   // === Motion positions (generated from XML) START ===
   ACTUAL_CHOOSEN_TYPE.Motion.Gluing_Nozzle_Z.Position[1].Pos := 143.76;
   ACTUAL_CHOOSEN_TYPE.Motion.Gluing_Nozzle_Z.Position[1].Vel := 200;
   ACTUAL_CHOOSEN_TYPE.Motion.Gluing_Nozzle_Z.Position[2].Pos := 139.11;
   ACTUAL_CHOOSEN_TYPE.Motion.Gluing_Nozzle_Z.Position[2].Vel := 200;
   ACTUAL_CHOOSEN_TYPE.Motion.Gluing_Nozzle_Z.Position[3].Pos := 131.98;
   ACTUAL_CHOOSEN_TYPE.Motion.Gluing_Nozzle_Z.Position[3].Vel := 200;
   ACTUAL_CHOOSEN_TYPE.Motion.Gluing_Nozzle_Z.Position[4].Pos := 127.89;
   ACTUAL_CHOOSEN_TYPE.Motion.Gluing_Nozzle_Z.Position[4].Vel := 200;
   ACTUAL_CHOOSEN_TYPE.Motion.Gluing_Nozzle_Z.Position[5].Pos := 0.0;
   ACTUAL_CHOOSEN_TYPE.Motion.Gluing_Nozzle_Z.Position[5].Vel := 0;
   ACTUAL_CHOOSEN_TYPE.Motion.Gluing_Nozzle_Z.Position[6].Pos := 127.0;
   ACTUAL_CHOOSEN_TYPE.Motion.Gluing_Nozzle_Z.Position[6].Vel := 200;
   ACTUAL_CHOOSEN_TYPE.Motion.Gluing_Nozzle_Z.Position[7].Pos := 48.11;
   ACTUAL_CHOOSEN_TYPE.Motion.Gluing_Nozzle_Z.Position[7].Vel := 200;
   ACTUAL_CHOOSEN_TYPE.Motion.Gluing_Nozzle_Z.Position[8].Pos := 0.0;
   ACTUAL_CHOOSEN_TYPE.Motion.Gluing_Nozzle_Z.Position[8].Vel := 200;
   ACTUAL_CHOOSEN_TYPE.Motion.Gluing_Nozzle_Z.Position[9].Pos := 123.0;
   ACTUAL_CHOOSEN_TYPE.Motion.Gluing_Nozzle_Z.Position[9].Vel := 200;
   ACTUAL_CHOOSEN_TYPE.Motion.Gluing_Nozzle_Z.Position[10].Pos := 0.0;
   ACTUAL_CHOOSEN_TYPE.Motion.Gluing_Nozzle_Z.Position[10].Vel := 0;
   ACTUAL_CHOOSEN_TYPE.Motion.Gluing_Nozzle_Z.Position[11].Pos := 0.0;
   ACTUAL_CHOOSEN_TYPE.Motion.Gluing_Nozzle_Z.Position[11].Vel := 0;
   ACTUAL_CHOOSEN_TYPE.Motion.Gluing_Nozzle_Z.Position[12].Pos := 0.0;
   ACTUAL_CHOOSEN_TYPE.Motion.Gluing_Nozzle_Z.Position[12].Vel := 0;
   ACTUAL_CHOOSEN_TYPE.Motion.Gluing_Nozzle_Z.Position[13].Pos := 0.0;
   ACTUAL_CHOOSEN_TYPE.Motion.Gluing_Nozzle_Z.Position[13].Vel := 0;
   ACTUAL_CHOOSEN_TYPE.Motion.Gluing_Nozzle_Z.Position[14].Pos := 0.0;
   ACTUAL_CHOOSEN_TYPE.Motion.Gluing_Nozzle_Z.Position[14].Vel := 0;
   ACTUAL_CHOOSEN_TYPE.Motion.Gluing_Nozzle_Z.Position[15].Pos := 0.0;
   ACTUAL_CHOOSEN_TYPE.Motion.Gluing_Nozzle_Z.Position[15].Vel := 0;
   ACTUAL_CHOOSEN_TYPE.Motion.Gluing_Nozzle_Z.Position[16].Pos := 0.0;
   ACTUAL_CHOOSEN_TYPE.Motion.Gluing_Nozzle_Z.Position[16].Vel := 0;
   ACTUAL_CHOOSEN_TYPE.Motion.Gluing_Nozzle_Z.Position[17].Pos := 0.0;
   ACTUAL_CHOOSEN_TYPE.Motion.Gluing_Nozzle_Z.Position[17].Vel := 0;
   ACTUAL_CHOOSEN_TYPE.Motion.Gluing_Nozzle_Z.Position[18].Pos := 0.0;
   ACTUAL_CHOOSEN_TYPE.Motion.Gluing_Nozzle_Z.Position[18].Vel := 0;
   ACTUAL_CHOOSEN_TYPE.Motion.Gluing_Nozzle_Z.Position[19].Pos := 0.0;
   ACTUAL_CHOOSEN_TYPE.Motion.Gluing_Nozzle_Z.Position[19].Vel := 0;
   ACTUAL_CHOOSEN_TYPE.Motion.Gluing_Nozzle_Z.Position[20].Pos := 0.0;
   ACTUAL_CHOOSEN_TYPE.Motion.Gluing_Nozzle_Z.Position[20].Vel := 0;
   ACTUAL_CHOOSEN_TYPE.Motion.Gluing_Nozzle_X.Position[1].Pos := 2.34;
   ACTUAL_CHOOSEN_TYPE.Motion.Gluing_Nozzle_X.Position[1].Vel := 200;
   ACTUAL_CHOOSEN_TYPE.Motion.Gluing_Nozzle_X.Position[2].Pos := 76.0;
   ACTUAL_CHOOSEN_TYPE.Motion.Gluing_Nozzle_X.Position[2].Vel := 200;
   ACTUAL_CHOOSEN_TYPE.Motion.Gluing_Nozzle_X.Position[3].Pos := 84.69;
   ACTUAL_CHOOSEN_TYPE.Motion.Gluing_Nozzle_X.Position[3].Vel := 200;
   ACTUAL_CHOOSEN_TYPE.Motion.Gluing_Nozzle_X.Position[4].Pos := 84.69;
   ACTUAL_CHOOSEN_TYPE.Motion.Gluing_Nozzle_X.Position[4].Vel := 200;
   ACTUAL_CHOOSEN_TYPE.Motion.Gluing_Nozzle_X.Position[5].Pos := 84.69;
   ACTUAL_CHOOSEN_TYPE.Motion.Gluing_Nozzle_X.Position[5].Vel := 200;
   ACTUAL_CHOOSEN_TYPE.Motion.Gluing_Nozzle_X.Position[6].Pos := 84.69;
   ACTUAL_CHOOSEN_TYPE.Motion.Gluing_Nozzle_X.Position[6].Vel := 200;
   ACTUAL_CHOOSEN_TYPE.Motion.Gluing_Nozzle_X.Position[7].Pos := 85.0;
   ACTUAL_CHOOSEN_TYPE.Motion.Gluing_Nozzle_X.Position[7].Vel := 200;
   ACTUAL_CHOOSEN_TYPE.Motion.Gluing_Nozzle_X.Position[8].Pos := 88.53;
   ACTUAL_CHOOSEN_TYPE.Motion.Gluing_Nozzle_X.Position[8].Vel := 200;
   ACTUAL_CHOOSEN_TYPE.Motion.Gluing_Nozzle_X.Position[9].Pos := 0.0;
   ACTUAL_CHOOSEN_TYPE.Motion.Gluing_Nozzle_X.Position[9].Vel := 0;
   ACTUAL_CHOOSEN_TYPE.Motion.Gluing_Nozzle_X.Position[10].Pos := 0.0;
   ACTUAL_CHOOSEN_TYPE.Motion.Gluing_Nozzle_X.Position[10].Vel := 0;
   ACTUAL_CHOOSEN_TYPE.Motion.Gluing_Nozzle_X.Position[11].Pos := 0.0;
   ACTUAL_CHOOSEN_TYPE.Motion.Gluing_Nozzle_X.Position[11].Vel := 0;
   ACTUAL_CHOOSEN_TYPE.Motion.Gluing_Nozzle_X.Position[12].Pos := 0.0;
   ACTUAL_CHOOSEN_TYPE.Motion.Gluing_Nozzle_X.Position[12].Vel := 0;
   ACTUAL_CHOOSEN_TYPE.Motion.Gluing_Nozzle_X.Position[13].Pos := 0.0;
   ACTUAL_CHOOSEN_TYPE.Motion.Gluing_Nozzle_X.Position[13].Vel := 0;
   ACTUAL_CHOOSEN_TYPE.Motion.Gluing_Nozzle_X.Position[14].Pos := 0.0;
   ACTUAL_CHOOSEN_TYPE.Motion.Gluing_Nozzle_X.Position[14].Vel := 0;
   ACTUAL_CHOOSEN_TYPE.Motion.Gluing_Nozzle_X.Position[15].Pos := 0.0;
   ACTUAL_CHOOSEN_TYPE.Motion.Gluing_Nozzle_X.Position[15].Vel := 0;
   ACTUAL_CHOOSEN_TYPE.Motion.Gluing_Nozzle_X.Position[16].Pos := 0.0;
   ACTUAL_CHOOSEN_TYPE.Motion.Gluing_Nozzle_X.Position[16].Vel := 0;
   ACTUAL_CHOOSEN_TYPE.Motion.Gluing_Nozzle_X.Position[17].Pos := 0.0;
   ACTUAL_CHOOSEN_TYPE.Motion.Gluing_Nozzle_X.Position[17].Vel := 0;
   ACTUAL_CHOOSEN_TYPE.Motion.Gluing_Nozzle_X.Position[18].Pos := 0.0;
   ACTUAL_CHOOSEN_TYPE.Motion.Gluing_Nozzle_X.Position[18].Vel := 0;
   ACTUAL_CHOOSEN_TYPE.Motion.Gluing_Nozzle_X.Position[19].Pos := 0.0;
   ACTUAL_CHOOSEN_TYPE.Motion.Gluing_Nozzle_X.Position[19].Vel := 0;
   ACTUAL_CHOOSEN_TYPE.Motion.Gluing_Nozzle_X.Position[20].Pos := 0.0;
   ACTUAL_CHOOSEN_TYPE.Motion.Gluing_Nozzle_X.Position[20].Vel := 0;
   ACTUAL_CHOOSEN_TYPE.Motion.Gluing_Nozzle_Y.Position[1].Pos := 115.47;
   ACTUAL_CHOOSEN_TYPE.Motion.Gluing_Nozzle_Y.Position[1].Vel := 200;
   ACTUAL_CHOOSEN_TYPE.Motion.Gluing_Nozzle_Y.Position[2].Pos := 115.47;
   ACTUAL_CHOOSEN_TYPE.Motion.Gluing_Nozzle_Y.Position[2].Vel := 200;
   ACTUAL_CHOOSEN_TYPE.Motion.Gluing_Nozzle_Y.Position[3].Pos := 115.47;
   ACTUAL_CHOOSEN_TYPE.Motion.Gluing_Nozzle_Y.Position[3].Vel := 200;
   ACTUAL_CHOOSEN_TYPE.Motion.Gluing_Nozzle_Y.Position[4].Pos := 115.47;
   ACTUAL_CHOOSEN_TYPE.Motion.Gluing_Nozzle_Y.Position[4].Vel := 200;
   ACTUAL_CHOOSEN_TYPE.Motion.Gluing_Nozzle_Y.Position[5].Pos := 115.47;
   ACTUAL_CHOOSEN_TYPE.Motion.Gluing_Nozzle_Y.Position[5].Vel := 200;
   ACTUAL_CHOOSEN_TYPE.Motion.Gluing_Nozzle_Y.Position[6].Pos := 110.18;
   ACTUAL_CHOOSEN_TYPE.Motion.Gluing_Nozzle_Y.Position[6].Vel := 200;
   ACTUAL_CHOOSEN_TYPE.Motion.Gluing_Nozzle_Y.Position[7].Pos := 60.52;
   ACTUAL_CHOOSEN_TYPE.Motion.Gluing_Nozzle_Y.Position[7].Vel := 200;
   ACTUAL_CHOOSEN_TYPE.Motion.Gluing_Nozzle_Y.Position[8].Pos := 80.0;
   ACTUAL_CHOOSEN_TYPE.Motion.Gluing_Nozzle_Y.Position[8].Vel := 100;
   ACTUAL_CHOOSEN_TYPE.Motion.Gluing_Nozzle_Y.Position[9].Pos := 0.0;
   ACTUAL_CHOOSEN_TYPE.Motion.Gluing_Nozzle_Y.Position[9].Vel := 0;
   ACTUAL_CHOOSEN_TYPE.Motion.Gluing_Nozzle_Y.Position[10].Pos := 0.0;
   ACTUAL_CHOOSEN_TYPE.Motion.Gluing_Nozzle_Y.Position[10].Vel := 0;
   ACTUAL_CHOOSEN_TYPE.Motion.Gluing_Nozzle_Y.Position[11].Pos := 0.0;
   ACTUAL_CHOOSEN_TYPE.Motion.Gluing_Nozzle_Y.Position[11].Vel := 0;
   ACTUAL_CHOOSEN_TYPE.Motion.Gluing_Nozzle_Y.Position[12].Pos := 0.0;
   ACTUAL_CHOOSEN_TYPE.Motion.Gluing_Nozzle_Y.Position[12].Vel := 0;
   ACTUAL_CHOOSEN_TYPE.Motion.Gluing_Nozzle_Y.Position[13].Pos := 0.0;
   ACTUAL_CHOOSEN_TYPE.Motion.Gluing_Nozzle_Y.Position[13].Vel := 0;
   ACTUAL_CHOOSEN_TYPE.Motion.Gluing_Nozzle_Y.Position[14].Pos := 0.0;
   ACTUAL_CHOOSEN_TYPE.Motion.Gluing_Nozzle_Y.Position[14].Vel := 0;
   ACTUAL_CHOOSEN_TYPE.Motion.Gluing_Nozzle_Y.Position[15].Pos := 0.0;
   ACTUAL_CHOOSEN_TYPE.Motion.Gluing_Nozzle_Y.Position[15].Vel := 0;
   ACTUAL_CHOOSEN_TYPE.Motion.Gluing_Nozzle_Y.Position[16].Pos := 0.0;
   ACTUAL_CHOOSEN_TYPE.Motion.Gluing_Nozzle_Y.Position[16].Vel := 0;
   ACTUAL_CHOOSEN_TYPE.Motion.Gluing_Nozzle_Y.Position[17].Pos := 0.0;
   ACTUAL_CHOOSEN_TYPE.Motion.Gluing_Nozzle_Y.Position[17].Vel := 0;
   ACTUAL_CHOOSEN_TYPE.Motion.Gluing_Nozzle_Y.Position[18].Pos := 0.0;
   ACTUAL_CHOOSEN_TYPE.Motion.Gluing_Nozzle_Y.Position[18].Vel := 0;
   ACTUAL_CHOOSEN_TYPE.Motion.Gluing_Nozzle_Y.Position[19].Pos := 0.0;
   ACTUAL_CHOOSEN_TYPE.Motion.Gluing_Nozzle_Y.Position[19].Vel := 0;
   ACTUAL_CHOOSEN_TYPE.Motion.Gluing_Nozzle_Y.Position[20].Pos := 0.0;
   ACTUAL_CHOOSEN_TYPE.Motion.Gluing_Nozzle_Y.Position[20].Vel := 0;
   ACTUAL_CHOOSEN_TYPE.Motion.Ring_Turntable_Axis_1.Position[1].Pos := 3419;
   ACTUAL_CHOOSEN_TYPE.Motion.Ring_Turntable_Axis_1.Position[1].Vel := 10000;
   ACTUAL_CHOOSEN_TYPE.Motion.Ring_Turntable_Axis_1.Position[2].Pos := 48386;
   ACTUAL_CHOOSEN_TYPE.Motion.Ring_Turntable_Axis_1.Position[2].Vel := 10000;
   ACTUAL_CHOOSEN_TYPE.Motion.Ring_Turntable_Axis_1.Position[3].Pos := 93294;
   ACTUAL_CHOOSEN_TYPE.Motion.Ring_Turntable_Axis_1.Position[3].Vel := 10000;
   ACTUAL_CHOOSEN_TYPE.Motion.Ring_Turntable_Axis_1.Position[4].Pos := 138335;
   ACTUAL_CHOOSEN_TYPE.Motion.Ring_Turntable_Axis_1.Position[4].Vel := 10000;
   ACTUAL_CHOOSEN_TYPE.Motion.Ring_Turntable_Axis_1.Position[5].Pos := 183464;
   ACTUAL_CHOOSEN_TYPE.Motion.Ring_Turntable_Axis_1.Position[5].Vel := 10000;
   ACTUAL_CHOOSEN_TYPE.Motion.Ring_Turntable_Axis_1.Position[6].Pos := 228443;
   ACTUAL_CHOOSEN_TYPE.Motion.Ring_Turntable_Axis_1.Position[6].Vel := 10000;
   ACTUAL_CHOOSEN_TYPE.Motion.Ring_Turntable_Axis_1.Position[7].Pos := 273535;
   ACTUAL_CHOOSEN_TYPE.Motion.Ring_Turntable_Axis_1.Position[7].Vel := 10000;
   ACTUAL_CHOOSEN_TYPE.Motion.Ring_Turntable_Axis_1.Position[8].Pos := 318250;
   ACTUAL_CHOOSEN_TYPE.Motion.Ring_Turntable_Axis_1.Position[8].Vel := 10000;
   ACTUAL_CHOOSEN_TYPE.Motion.Ring_Turntable_Axis_1.Position[9].Pos := 0;
   ACTUAL_CHOOSEN_TYPE.Motion.Ring_Turntable_Axis_1.Position[9].Vel := 0;
   ACTUAL_CHOOSEN_TYPE.Motion.Ring_Turntable_Axis_1.Position[10].Pos := 0;
   ACTUAL_CHOOSEN_TYPE.Motion.Ring_Turntable_Axis_1.Position[10].Vel := 0;
   ACTUAL_CHOOSEN_TYPE.Motion.Ring_Turntable_Axis_1.Position[11].Pos := 0;
   ACTUAL_CHOOSEN_TYPE.Motion.Ring_Turntable_Axis_1.Position[11].Vel := 0;
   ACTUAL_CHOOSEN_TYPE.Motion.Ring_Turntable_Axis_1.Position[12].Pos := 0;
   ACTUAL_CHOOSEN_TYPE.Motion.Ring_Turntable_Axis_1.Position[12].Vel := 0;
   ACTUAL_CHOOSEN_TYPE.Motion.Ring_Turntable_Axis_1.Position[13].Pos := 0;
   ACTUAL_CHOOSEN_TYPE.Motion.Ring_Turntable_Axis_1.Position[13].Vel := 0;
   ACTUAL_CHOOSEN_TYPE.Motion.Ring_Turntable_Axis_1.Position[14].Pos := 0;
   ACTUAL_CHOOSEN_TYPE.Motion.Ring_Turntable_Axis_1.Position[14].Vel := 0;
   ACTUAL_CHOOSEN_TYPE.Motion.Ring_Turntable_Axis_1.Position[15].Pos := 0;
   ACTUAL_CHOOSEN_TYPE.Motion.Ring_Turntable_Axis_1.Position[15].Vel := 0;
   ACTUAL_CHOOSEN_TYPE.Motion.Ring_Turntable_Axis_1.Position[16].Pos := 0;
   ACTUAL_CHOOSEN_TYPE.Motion.Ring_Turntable_Axis_1.Position[16].Vel := 0;
   ACTUAL_CHOOSEN_TYPE.Motion.Ring_Turntable_Axis_1.Position[17].Pos := 0;
   ACTUAL_CHOOSEN_TYPE.Motion.Ring_Turntable_Axis_1.Position[17].Vel := 0;
   ACTUAL_CHOOSEN_TYPE.Motion.Ring_Turntable_Axis_1.Position[18].Pos := 0;
   ACTUAL_CHOOSEN_TYPE.Motion.Ring_Turntable_Axis_1.Position[18].Vel := 0;
   ACTUAL_CHOOSEN_TYPE.Motion.Ring_Turntable_Axis_1.Position[19].Pos := 0;
   ACTUAL_CHOOSEN_TYPE.Motion.Ring_Turntable_Axis_1.Position[19].Vel := 0;
   ACTUAL_CHOOSEN_TYPE.Motion.Ring_Turntable_Axis_1.Position[20].Pos := 0;
   ACTUAL_CHOOSEN_TYPE.Motion.Ring_Turntable_Axis_1.Position[20].Vel := 0;
   ACTUAL_CHOOSEN_TYPE.Motion.Shaft_Scan_Turntable_Axis.Position[1].Pos := 0;
   ACTUAL_CHOOSEN_TYPE.Motion.Shaft_Scan_Turntable_Axis.Position[1].Vel := 10000;
   ACTUAL_CHOOSEN_TYPE.Motion.Shaft_Scan_Turntable_Axis.Position[2].Pos := 450000;
   ACTUAL_CHOOSEN_TYPE.Motion.Shaft_Scan_Turntable_Axis.Position[2].Vel := 10000;
   ACTUAL_CHOOSEN_TYPE.Motion.Shaft_Scan_Turntable_Axis.Position[3].Pos := 900000;
   ACTUAL_CHOOSEN_TYPE.Motion.Shaft_Scan_Turntable_Axis.Position[3].Vel := 10000;
   ACTUAL_CHOOSEN_TYPE.Motion.Shaft_Scan_Turntable_Axis.Position[4].Pos := 135000;
   ACTUAL_CHOOSEN_TYPE.Motion.Shaft_Scan_Turntable_Axis.Position[4].Vel := 10000;
   ACTUAL_CHOOSEN_TYPE.Motion.Shaft_Scan_Turntable_Axis.Position[5].Pos := 180000;
   ACTUAL_CHOOSEN_TYPE.Motion.Shaft_Scan_Turntable_Axis.Position[5].Vel := 10000;
   ACTUAL_CHOOSEN_TYPE.Motion.Shaft_Scan_Turntable_Axis.Position[6].Pos := 225000;
   ACTUAL_CHOOSEN_TYPE.Motion.Shaft_Scan_Turntable_Axis.Position[6].Vel := 10000;
   ACTUAL_CHOOSEN_TYPE.Motion.Shaft_Scan_Turntable_Axis.Position[7].Pos := 270000;
   ACTUAL_CHOOSEN_TYPE.Motion.Shaft_Scan_Turntable_Axis.Position[7].Vel := 10000;
   ACTUAL_CHOOSEN_TYPE.Motion.Shaft_Scan_Turntable_Axis.Position[8].Pos := 315000;
   ACTUAL_CHOOSEN_TYPE.Motion.Shaft_Scan_Turntable_Axis.Position[8].Vel := 10000;
   ACTUAL_CHOOSEN_TYPE.Motion.Shaft_Scan_Turntable_Axis.Position[9].Pos := 0;
   ACTUAL_CHOOSEN_TYPE.Motion.Shaft_Scan_Turntable_Axis.Position[9].Vel := 0;
   ACTUAL_CHOOSEN_TYPE.Motion.Shaft_Scan_Turntable_Axis.Position[10].Pos := 0;
   ACTUAL_CHOOSEN_TYPE.Motion.Shaft_Scan_Turntable_Axis.Position[10].Vel := 0;
   ACTUAL_CHOOSEN_TYPE.Motion.Shaft_Scan_Turntable_Axis.Position[11].Pos := 0;
   ACTUAL_CHOOSEN_TYPE.Motion.Shaft_Scan_Turntable_Axis.Position[11].Vel := 0;
   ACTUAL_CHOOSEN_TYPE.Motion.Shaft_Scan_Turntable_Axis.Position[12].Pos := 0;
   ACTUAL_CHOOSEN_TYPE.Motion.Shaft_Scan_Turntable_Axis.Position[12].Vel := 0;
   ACTUAL_CHOOSEN_TYPE.Motion.Shaft_Scan_Turntable_Axis.Position[13].Pos := 0;
   ACTUAL_CHOOSEN_TYPE.Motion.Shaft_Scan_Turntable_Axis.Position[13].Vel := 0;
   ACTUAL_CHOOSEN_TYPE.Motion.Shaft_Scan_Turntable_Axis.Position[14].Pos := 0;
   ACTUAL_CHOOSEN_TYPE.Motion.Shaft_Scan_Turntable_Axis.Position[14].Vel := 0;
   ACTUAL_CHOOSEN_TYPE.Motion.Shaft_Scan_Turntable_Axis.Position[15].Pos := 0;
   ACTUAL_CHOOSEN_TYPE.Motion.Shaft_Scan_Turntable_Axis.Position[15].Vel := 0;
   ACTUAL_CHOOSEN_TYPE.Motion.Shaft_Scan_Turntable_Axis.Position[16].Pos := 0;
   ACTUAL_CHOOSEN_TYPE.Motion.Shaft_Scan_Turntable_Axis.Position[16].Vel := 0;
   ACTUAL_CHOOSEN_TYPE.Motion.Shaft_Scan_Turntable_Axis.Position[17].Pos := 0;
   ACTUAL_CHOOSEN_TYPE.Motion.Shaft_Scan_Turntable_Axis.Position[17].Vel := 0;
   ACTUAL_CHOOSEN_TYPE.Motion.Shaft_Scan_Turntable_Axis.Position[18].Pos := 0;
   ACTUAL_CHOOSEN_TYPE.Motion.Shaft_Scan_Turntable_Axis.Position[18].Vel := 0;
   ACTUAL_CHOOSEN_TYPE.Motion.Shaft_Scan_Turntable_Axis.Position[19].Pos := 0;
   ACTUAL_CHOOSEN_TYPE.Motion.Shaft_Scan_Turntable_Axis.Position[19].Vel := 0;
   ACTUAL_CHOOSEN_TYPE.Motion.Shaft_Scan_Turntable_Axis.Position[20].Pos := 0;
   ACTUAL_CHOOSEN_TYPE.Motion.Shaft_Scan_Turntable_Axis.Position[20].Vel := 0;
   ACTUAL_CHOOSEN_TYPE.Motion.Gluing_Rotary_Jig_Axis.Position[1].Pos := 0;
   ACTUAL_CHOOSEN_TYPE.Motion.Gluing_Rotary_Jig_Axis.Position[1].Vel := 20000;
   ACTUAL_CHOOSEN_TYPE.Motion.Gluing_Rotary_Jig_Axis.Position[2].Pos := 0;
   ACTUAL_CHOOSEN_TYPE.Motion.Gluing_Rotary_Jig_Axis.Position[2].Vel := 20000;
   ACTUAL_CHOOSEN_TYPE.Motion.Gluing_Rotary_Jig_Axis.Position[3].Pos := 680000;
   ACTUAL_CHOOSEN_TYPE.Motion.Gluing_Rotary_Jig_Axis.Position[3].Vel := 10000;
   ACTUAL_CHOOSEN_TYPE.Motion.Gluing_Rotary_Jig_Axis.Position[4].Pos := 680000;
   ACTUAL_CHOOSEN_TYPE.Motion.Gluing_Rotary_Jig_Axis.Position[4].Vel := 10000;
   ACTUAL_CHOOSEN_TYPE.Motion.Gluing_Rotary_Jig_Axis.Position[5].Pos := 680000;
   ACTUAL_CHOOSEN_TYPE.Motion.Gluing_Rotary_Jig_Axis.Position[5].Vel := 10000;
   ACTUAL_CHOOSEN_TYPE.Motion.Gluing_Rotary_Jig_Axis.Position[6].Pos := 680000;
   ACTUAL_CHOOSEN_TYPE.Motion.Gluing_Rotary_Jig_Axis.Position[6].Vel := 10000;
   ACTUAL_CHOOSEN_TYPE.Motion.Gluing_Rotary_Jig_Axis.Position[7].Pos := 90000;
   ACTUAL_CHOOSEN_TYPE.Motion.Gluing_Rotary_Jig_Axis.Position[7].Vel := 10000;
   ACTUAL_CHOOSEN_TYPE.Motion.Gluing_Rotary_Jig_Axis.Position[8].Pos := 180000;
   ACTUAL_CHOOSEN_TYPE.Motion.Gluing_Rotary_Jig_Axis.Position[8].Vel := 10000;
   ACTUAL_CHOOSEN_TYPE.Motion.Gluing_Rotary_Jig_Axis.Position[9].Pos := 270000;
   ACTUAL_CHOOSEN_TYPE.Motion.Gluing_Rotary_Jig_Axis.Position[9].Vel := 10000;
   ACTUAL_CHOOSEN_TYPE.Motion.Gluing_Rotary_Jig_Axis.Position[10].Pos := 0;
   ACTUAL_CHOOSEN_TYPE.Motion.Gluing_Rotary_Jig_Axis.Position[10].Vel := 0;
   ACTUAL_CHOOSEN_TYPE.Motion.Gluing_Rotary_Jig_Axis.Position[11].Pos := 0;
   ACTUAL_CHOOSEN_TYPE.Motion.Gluing_Rotary_Jig_Axis.Position[11].Vel := 0;
   ACTUAL_CHOOSEN_TYPE.Motion.Gluing_Rotary_Jig_Axis.Position[12].Pos := 0;
   ACTUAL_CHOOSEN_TYPE.Motion.Gluing_Rotary_Jig_Axis.Position[12].Vel := 0;
   ACTUAL_CHOOSEN_TYPE.Motion.Gluing_Rotary_Jig_Axis.Position[13].Pos := 0;
   ACTUAL_CHOOSEN_TYPE.Motion.Gluing_Rotary_Jig_Axis.Position[13].Vel := 0;
   ACTUAL_CHOOSEN_TYPE.Motion.Gluing_Rotary_Jig_Axis.Position[14].Pos := 0;
   ACTUAL_CHOOSEN_TYPE.Motion.Gluing_Rotary_Jig_Axis.Position[14].Vel := 0;
   ACTUAL_CHOOSEN_TYPE.Motion.Gluing_Rotary_Jig_Axis.Position[15].Pos := 0;
   ACTUAL_CHOOSEN_TYPE.Motion.Gluing_Rotary_Jig_Axis.Position[15].Vel := 0;
   ACTUAL_CHOOSEN_TYPE.Motion.Gluing_Rotary_Jig_Axis.Position[16].Pos := 0;
   ACTUAL_CHOOSEN_TYPE.Motion.Gluing_Rotary_Jig_Axis.Position[16].Vel := 0;
   ACTUAL_CHOOSEN_TYPE.Motion.Gluing_Rotary_Jig_Axis.Position[17].Pos := 0;
   ACTUAL_CHOOSEN_TYPE.Motion.Gluing_Rotary_Jig_Axis.Position[17].Vel := 0;
   ACTUAL_CHOOSEN_TYPE.Motion.Gluing_Rotary_Jig_Axis.Position[18].Pos := 0;
   ACTUAL_CHOOSEN_TYPE.Motion.Gluing_Rotary_Jig_Axis.Position[18].Vel := 0;
   ACTUAL_CHOOSEN_TYPE.Motion.Gluing_Rotary_Jig_Axis.Position[19].Pos := 0;
   ACTUAL_CHOOSEN_TYPE.Motion.Gluing_Rotary_Jig_Axis.Position[19].Vel := 0;
   ACTUAL_CHOOSEN_TYPE.Motion.Gluing_Rotary_Jig_Axis.Position[20].Pos := 0;
   ACTUAL_CHOOSEN_TYPE.Motion.Gluing_Rotary_Jig_Axis.Position[20].Vel := 0;
   ACTUAL_CHOOSEN_TYPE.Motion.Ring_Turntable_Axis_2.Position[1].Pos := 3585;
   ACTUAL_CHOOSEN_TYPE.Motion.Ring_Turntable_Axis_2.Position[1].Vel := 10000;
   ACTUAL_CHOOSEN_TYPE.Motion.Ring_Turntable_Axis_2.Position[2].Pos := 48610;
   ACTUAL_CHOOSEN_TYPE.Motion.Ring_Turntable_Axis_2.Position[2].Vel := 10000;
   ACTUAL_CHOOSEN_TYPE.Motion.Ring_Turntable_Axis_2.Position[3].Pos := 93637;
   ACTUAL_CHOOSEN_TYPE.Motion.Ring_Turntable_Axis_2.Position[3].Vel := 10000;
   ACTUAL_CHOOSEN_TYPE.Motion.Ring_Turntable_Axis_2.Position[4].Pos := 138606;
   ACTUAL_CHOOSEN_TYPE.Motion.Ring_Turntable_Axis_2.Position[4].Vel := 10000;
   ACTUAL_CHOOSEN_TYPE.Motion.Ring_Turntable_Axis_2.Position[5].Pos := 183388;
   ACTUAL_CHOOSEN_TYPE.Motion.Ring_Turntable_Axis_2.Position[5].Vel := 10000;
   ACTUAL_CHOOSEN_TYPE.Motion.Ring_Turntable_Axis_2.Position[6].Pos := 228458;
   ACTUAL_CHOOSEN_TYPE.Motion.Ring_Turntable_Axis_2.Position[6].Vel := 10000;
   ACTUAL_CHOOSEN_TYPE.Motion.Ring_Turntable_Axis_2.Position[7].Pos := 273513;
   ACTUAL_CHOOSEN_TYPE.Motion.Ring_Turntable_Axis_2.Position[7].Vel := 10000;
   ACTUAL_CHOOSEN_TYPE.Motion.Ring_Turntable_Axis_2.Position[8].Pos := 318501;
   ACTUAL_CHOOSEN_TYPE.Motion.Ring_Turntable_Axis_2.Position[8].Vel := 10000;
   ACTUAL_CHOOSEN_TYPE.Motion.Ring_Turntable_Axis_2.Position[9].Pos := 0;
   ACTUAL_CHOOSEN_TYPE.Motion.Ring_Turntable_Axis_2.Position[9].Vel := 0;
   ACTUAL_CHOOSEN_TYPE.Motion.Ring_Turntable_Axis_2.Position[10].Pos := 0;
   ACTUAL_CHOOSEN_TYPE.Motion.Ring_Turntable_Axis_2.Position[10].Vel := 0;
   ACTUAL_CHOOSEN_TYPE.Motion.Ring_Turntable_Axis_2.Position[11].Pos := 0;
   ACTUAL_CHOOSEN_TYPE.Motion.Ring_Turntable_Axis_2.Position[11].Vel := 0;
   ACTUAL_CHOOSEN_TYPE.Motion.Ring_Turntable_Axis_2.Position[12].Pos := 0;
   ACTUAL_CHOOSEN_TYPE.Motion.Ring_Turntable_Axis_2.Position[12].Vel := 0;
   ACTUAL_CHOOSEN_TYPE.Motion.Ring_Turntable_Axis_2.Position[13].Pos := 0;
   ACTUAL_CHOOSEN_TYPE.Motion.Ring_Turntable_Axis_2.Position[13].Vel := 0;
   ACTUAL_CHOOSEN_TYPE.Motion.Ring_Turntable_Axis_2.Position[14].Pos := 0;
   ACTUAL_CHOOSEN_TYPE.Motion.Ring_Turntable_Axis_2.Position[14].Vel := 0;
   ACTUAL_CHOOSEN_TYPE.Motion.Ring_Turntable_Axis_2.Position[15].Pos := 0;
   ACTUAL_CHOOSEN_TYPE.Motion.Ring_Turntable_Axis_2.Position[15].Vel := 0;
   ACTUAL_CHOOSEN_TYPE.Motion.Ring_Turntable_Axis_2.Position[16].Pos := 0;
   ACTUAL_CHOOSEN_TYPE.Motion.Ring_Turntable_Axis_2.Position[16].Vel := 0;
   ACTUAL_CHOOSEN_TYPE.Motion.Ring_Turntable_Axis_2.Position[17].Pos := 0;
   ACTUAL_CHOOSEN_TYPE.Motion.Ring_Turntable_Axis_2.Position[17].Vel := 0;
   ACTUAL_CHOOSEN_TYPE.Motion.Ring_Turntable_Axis_2.Position[18].Pos := 0;
   ACTUAL_CHOOSEN_TYPE.Motion.Ring_Turntable_Axis_2.Position[18].Vel := 0;
   ACTUAL_CHOOSEN_TYPE.Motion.Ring_Turntable_Axis_2.Position[19].Pos := 0;
   ACTUAL_CHOOSEN_TYPE.Motion.Ring_Turntable_Axis_2.Position[19].Vel := 0;
   ACTUAL_CHOOSEN_TYPE.Motion.Ring_Turntable_Axis_2.Position[20].Pos := 0;
   ACTUAL_CHOOSEN_TYPE.Motion.Ring_Turntable_Axis_2.Position[20].Vel := 0;
   PRODUCT_TYPE[1].Motion.Gluing_Nozzle_Z.Position[1].Pos := 143.76;
   PRODUCT_TYPE[1].Motion.Gluing_Nozzle_Z.Position[1].Vel := 200;
   PRODUCT_TYPE[2].Motion.Gluing_Nozzle_Z.Position[1].Pos := 143.76;
   PRODUCT_TYPE[2].Motion.Gluing_Nozzle_Z.Position[1].Vel := 200;
   PRODUCT_TYPE[3].Motion.Gluing_Nozzle_Z.Position[1].Pos := 143.76;
   PRODUCT_TYPE[3].Motion.Gluing_Nozzle_Z.Position[1].Vel := 200;
   PRODUCT_TYPE[4].Motion.Gluing_Nozzle_Z.Position[1].Pos := 143.76;
   PRODUCT_TYPE[4].Motion.Gluing_Nozzle_Z.Position[1].Vel := 200;
   PRODUCT_TYPE[5].Motion.Gluing_Nozzle_Z.Position[1].Pos := 143.76;
   PRODUCT_TYPE[5].Motion.Gluing_Nozzle_Z.Position[1].Vel := 200;
   PRODUCT_TYPE[6].Motion.Gluing_Nozzle_Z.Position[1].Pos := 143.76;
   PRODUCT_TYPE[6].Motion.Gluing_Nozzle_Z.Position[1].Vel := 200;
   PRODUCT_TYPE[7].Motion.Gluing_Nozzle_Z.Position[1].Pos := 143.76;
   PRODUCT_TYPE[7].Motion.Gluing_Nozzle_Z.Position[1].Vel := 200;
   PRODUCT_TYPE[8].Motion.Gluing_Nozzle_Z.Position[1].Pos := 143.76;
   PRODUCT_TYPE[8].Motion.Gluing_Nozzle_Z.Position[1].Vel := 200;
   PRODUCT_TYPE[9].Motion.Gluing_Nozzle_Z.Position[1].Pos := 143.76;
   PRODUCT_TYPE[9].Motion.Gluing_Nozzle_Z.Position[1].Vel := 200;
   PRODUCT_TYPE[10].Motion.Gluing_Nozzle_Z.Position[1].Pos := 143.76;
   PRODUCT_TYPE[10].Motion.Gluing_Nozzle_Z.Position[1].Vel := 200;
   PRODUCT_TYPE[1].Motion.Gluing_Nozzle_Z.Position[2].Pos := 139.11;
   PRODUCT_TYPE[1].Motion.Gluing_Nozzle_Z.Position[2].Vel := 200;
   PRODUCT_TYPE[2].Motion.Gluing_Nozzle_Z.Position[2].Pos := 139.11;
   PRODUCT_TYPE[2].Motion.Gluing_Nozzle_Z.Position[2].Vel := 200;
   PRODUCT_TYPE[3].Motion.Gluing_Nozzle_Z.Position[2].Pos := 139.11;
   PRODUCT_TYPE[3].Motion.Gluing_Nozzle_Z.Position[2].Vel := 200;
   PRODUCT_TYPE[4].Motion.Gluing_Nozzle_Z.Position[2].Pos := 139.11;
   PRODUCT_TYPE[4].Motion.Gluing_Nozzle_Z.Position[2].Vel := 200;
   PRODUCT_TYPE[5].Motion.Gluing_Nozzle_Z.Position[2].Pos := 139.11;
   PRODUCT_TYPE[5].Motion.Gluing_Nozzle_Z.Position[2].Vel := 200;
   PRODUCT_TYPE[6].Motion.Gluing_Nozzle_Z.Position[2].Pos := 139.11;
   PRODUCT_TYPE[6].Motion.Gluing_Nozzle_Z.Position[2].Vel := 200;
   PRODUCT_TYPE[7].Motion.Gluing_Nozzle_Z.Position[2].Pos := 139.11;
   PRODUCT_TYPE[7].Motion.Gluing_Nozzle_Z.Position[2].Vel := 200;
   PRODUCT_TYPE[8].Motion.Gluing_Nozzle_Z.Position[2].Pos := 139.11;
   PRODUCT_TYPE[8].Motion.Gluing_Nozzle_Z.Position[2].Vel := 200;
   PRODUCT_TYPE[9].Motion.Gluing_Nozzle_Z.Position[2].Pos := 139.11;
   PRODUCT_TYPE[9].Motion.Gluing_Nozzle_Z.Position[2].Vel := 200;
   PRODUCT_TYPE[10].Motion.Gluing_Nozzle_Z.Position[2].Pos := 139.11;
   PRODUCT_TYPE[10].Motion.Gluing_Nozzle_Z.Position[2].Vel := 200;
   PRODUCT_TYPE[1].Motion.Gluing_Nozzle_Z.Position[3].Pos := 131.98;
   PRODUCT_TYPE[1].Motion.Gluing_Nozzle_Z.Position[3].Vel := 200;
   PRODUCT_TYPE[2].Motion.Gluing_Nozzle_Z.Position[3].Pos := 131.98;
   PRODUCT_TYPE[2].Motion.Gluing_Nozzle_Z.Position[3].Vel := 200;
   PRODUCT_TYPE[3].Motion.Gluing_Nozzle_Z.Position[3].Pos := 131.98;
   PRODUCT_TYPE[3].Motion.Gluing_Nozzle_Z.Position[3].Vel := 200;
   PRODUCT_TYPE[4].Motion.Gluing_Nozzle_Z.Position[3].Pos := 131.98;
   PRODUCT_TYPE[4].Motion.Gluing_Nozzle_Z.Position[3].Vel := 200;
   PRODUCT_TYPE[5].Motion.Gluing_Nozzle_Z.Position[3].Pos := 131.98;
   PRODUCT_TYPE[5].Motion.Gluing_Nozzle_Z.Position[3].Vel := 200;
   PRODUCT_TYPE[6].Motion.Gluing_Nozzle_Z.Position[3].Pos := 131.98;
   PRODUCT_TYPE[6].Motion.Gluing_Nozzle_Z.Position[3].Vel := 200;
   PRODUCT_TYPE[7].Motion.Gluing_Nozzle_Z.Position[3].Pos := 131.98;
   PRODUCT_TYPE[7].Motion.Gluing_Nozzle_Z.Position[3].Vel := 200;
   PRODUCT_TYPE[8].Motion.Gluing_Nozzle_Z.Position[3].Pos := 131.98;
   PRODUCT_TYPE[8].Motion.Gluing_Nozzle_Z.Position[3].Vel := 200;
   PRODUCT_TYPE[9].Motion.Gluing_Nozzle_Z.Position[3].Pos := 131.98;
   PRODUCT_TYPE[9].Motion.Gluing_Nozzle_Z.Position[3].Vel := 200;
   PRODUCT_TYPE[10].Motion.Gluing_Nozzle_Z.Position[3].Pos := 131.98;
   PRODUCT_TYPE[10].Motion.Gluing_Nozzle_Z.Position[3].Vel := 200;
   PRODUCT_TYPE[1].Motion.Gluing_Nozzle_Z.Position[4].Pos := 127.89;
   PRODUCT_TYPE[1].Motion.Gluing_Nozzle_Z.Position[4].Vel := 200;
   PRODUCT_TYPE[2].Motion.Gluing_Nozzle_Z.Position[4].Pos := 127.89;
   PRODUCT_TYPE[2].Motion.Gluing_Nozzle_Z.Position[4].Vel := 200;
   PRODUCT_TYPE[3].Motion.Gluing_Nozzle_Z.Position[4].Pos := 127.89;
   PRODUCT_TYPE[3].Motion.Gluing_Nozzle_Z.Position[4].Vel := 200;
   PRODUCT_TYPE[4].Motion.Gluing_Nozzle_Z.Position[4].Pos := 127.89;
   PRODUCT_TYPE[4].Motion.Gluing_Nozzle_Z.Position[4].Vel := 200;
   PRODUCT_TYPE[5].Motion.Gluing_Nozzle_Z.Position[4].Pos := 127.89;
   PRODUCT_TYPE[5].Motion.Gluing_Nozzle_Z.Position[4].Vel := 200;
   PRODUCT_TYPE[6].Motion.Gluing_Nozzle_Z.Position[4].Pos := 127.89;
   PRODUCT_TYPE[6].Motion.Gluing_Nozzle_Z.Position[4].Vel := 200;
   PRODUCT_TYPE[7].Motion.Gluing_Nozzle_Z.Position[4].Pos := 127.89;
   PRODUCT_TYPE[7].Motion.Gluing_Nozzle_Z.Position[4].Vel := 200;
   PRODUCT_TYPE[8].Motion.Gluing_Nozzle_Z.Position[4].Pos := 127.89;
   PRODUCT_TYPE[8].Motion.Gluing_Nozzle_Z.Position[4].Vel := 200;
   PRODUCT_TYPE[9].Motion.Gluing_Nozzle_Z.Position[4].Pos := 127.89;
   PRODUCT_TYPE[9].Motion.Gluing_Nozzle_Z.Position[4].Vel := 200;
   PRODUCT_TYPE[10].Motion.Gluing_Nozzle_Z.Position[4].Pos := 127.89;
   PRODUCT_TYPE[10].Motion.Gluing_Nozzle_Z.Position[4].Vel := 200;
   PRODUCT_TYPE[1].Motion.Gluing_Nozzle_Z.Position[5].Pos := 0.0;
   PRODUCT_TYPE[1].Motion.Gluing_Nozzle_Z.Position[5].Vel := 0;
   PRODUCT_TYPE[2].Motion.Gluing_Nozzle_Z.Position[5].Pos := 0.0;
   PRODUCT_TYPE[2].Motion.Gluing_Nozzle_Z.Position[5].Vel := 0;
   PRODUCT_TYPE[3].Motion.Gluing_Nozzle_Z.Position[5].Pos := 0.0;
   PRODUCT_TYPE[3].Motion.Gluing_Nozzle_Z.Position[5].Vel := 0;
   PRODUCT_TYPE[4].Motion.Gluing_Nozzle_Z.Position[5].Pos := 0.0;
   PRODUCT_TYPE[4].Motion.Gluing_Nozzle_Z.Position[5].Vel := 0;
   PRODUCT_TYPE[5].Motion.Gluing_Nozzle_Z.Position[5].Pos := 0.0;
   PRODUCT_TYPE[5].Motion.Gluing_Nozzle_Z.Position[5].Vel := 0;
   PRODUCT_TYPE[6].Motion.Gluing_Nozzle_Z.Position[5].Pos := 0.0;
   PRODUCT_TYPE[6].Motion.Gluing_Nozzle_Z.Position[5].Vel := 0;
   PRODUCT_TYPE[7].Motion.Gluing_Nozzle_Z.Position[5].Pos := 0.0;
   PRODUCT_TYPE[7].Motion.Gluing_Nozzle_Z.Position[5].Vel := 0;
   PRODUCT_TYPE[8].Motion.Gluing_Nozzle_Z.Position[5].Pos := 0.0;
   PRODUCT_TYPE[8].Motion.Gluing_Nozzle_Z.Position[5].Vel := 0;
   PRODUCT_TYPE[9].Motion.Gluing_Nozzle_Z.Position[5].Pos := 0.0;
   PRODUCT_TYPE[9].Motion.Gluing_Nozzle_Z.Position[5].Vel := 0;
   PRODUCT_TYPE[10].Motion.Gluing_Nozzle_Z.Position[5].Pos := 0.0;
   PRODUCT_TYPE[10].Motion.Gluing_Nozzle_Z.Position[5].Vel := 0;
   PRODUCT_TYPE[1].Motion.Gluing_Nozzle_Z.Position[6].Pos := 127.0;
   PRODUCT_TYPE[1].Motion.Gluing_Nozzle_Z.Position[6].Vel := 200;
   PRODUCT_TYPE[2].Motion.Gluing_Nozzle_Z.Position[6].Pos := 127.0;
   PRODUCT_TYPE[2].Motion.Gluing_Nozzle_Z.Position[6].Vel := 200;
   PRODUCT_TYPE[3].Motion.Gluing_Nozzle_Z.Position[6].Pos := 127.0;
   PRODUCT_TYPE[3].Motion.Gluing_Nozzle_Z.Position[6].Vel := 200;
   PRODUCT_TYPE[4].Motion.Gluing_Nozzle_Z.Position[6].Pos := 127.0;
   PRODUCT_TYPE[4].Motion.Gluing_Nozzle_Z.Position[6].Vel := 200;
   PRODUCT_TYPE[5].Motion.Gluing_Nozzle_Z.Position[6].Pos := 127.0;
   PRODUCT_TYPE[5].Motion.Gluing_Nozzle_Z.Position[6].Vel := 200;
   PRODUCT_TYPE[6].Motion.Gluing_Nozzle_Z.Position[6].Pos := 127.0;
   PRODUCT_TYPE[6].Motion.Gluing_Nozzle_Z.Position[6].Vel := 200;
   PRODUCT_TYPE[7].Motion.Gluing_Nozzle_Z.Position[6].Pos := 127.0;
   PRODUCT_TYPE[7].Motion.Gluing_Nozzle_Z.Position[6].Vel := 200;
   PRODUCT_TYPE[8].Motion.Gluing_Nozzle_Z.Position[6].Pos := 127.0;
   PRODUCT_TYPE[8].Motion.Gluing_Nozzle_Z.Position[6].Vel := 200;
   PRODUCT_TYPE[9].Motion.Gluing_Nozzle_Z.Position[6].Pos := 127.0;
   PRODUCT_TYPE[9].Motion.Gluing_Nozzle_Z.Position[6].Vel := 200;
   PRODUCT_TYPE[10].Motion.Gluing_Nozzle_Z.Position[6].Pos := 127.0;
   PRODUCT_TYPE[10].Motion.Gluing_Nozzle_Z.Position[6].Vel := 200;
   PRODUCT_TYPE[1].Motion.Gluing_Nozzle_Z.Position[7].Pos := 48.11;
   PRODUCT_TYPE[1].Motion.Gluing_Nozzle_Z.Position[7].Vel := 200;
   PRODUCT_TYPE[2].Motion.Gluing_Nozzle_Z.Position[7].Pos := 48.11;
   PRODUCT_TYPE[2].Motion.Gluing_Nozzle_Z.Position[7].Vel := 200;
   PRODUCT_TYPE[3].Motion.Gluing_Nozzle_Z.Position[7].Pos := 48.11;
   PRODUCT_TYPE[3].Motion.Gluing_Nozzle_Z.Position[7].Vel := 200;
   PRODUCT_TYPE[4].Motion.Gluing_Nozzle_Z.Position[7].Pos := 48.11;
   PRODUCT_TYPE[4].Motion.Gluing_Nozzle_Z.Position[7].Vel := 200;
   PRODUCT_TYPE[5].Motion.Gluing_Nozzle_Z.Position[7].Pos := 48.11;
   PRODUCT_TYPE[5].Motion.Gluing_Nozzle_Z.Position[7].Vel := 200;
   PRODUCT_TYPE[6].Motion.Gluing_Nozzle_Z.Position[7].Pos := 48.11;
   PRODUCT_TYPE[6].Motion.Gluing_Nozzle_Z.Position[7].Vel := 200;
   PRODUCT_TYPE[7].Motion.Gluing_Nozzle_Z.Position[7].Pos := 48.11;
   PRODUCT_TYPE[7].Motion.Gluing_Nozzle_Z.Position[7].Vel := 200;
   PRODUCT_TYPE[8].Motion.Gluing_Nozzle_Z.Position[7].Pos := 48.11;
   PRODUCT_TYPE[8].Motion.Gluing_Nozzle_Z.Position[7].Vel := 200;
   PRODUCT_TYPE[9].Motion.Gluing_Nozzle_Z.Position[7].Pos := 48.11;
   PRODUCT_TYPE[9].Motion.Gluing_Nozzle_Z.Position[7].Vel := 200;
   PRODUCT_TYPE[10].Motion.Gluing_Nozzle_Z.Position[7].Pos := 48.11;
   PRODUCT_TYPE[10].Motion.Gluing_Nozzle_Z.Position[7].Vel := 200;
   PRODUCT_TYPE[1].Motion.Gluing_Nozzle_Z.Position[8].Pos := 0.0;
   PRODUCT_TYPE[1].Motion.Gluing_Nozzle_Z.Position[8].Vel := 200;
   PRODUCT_TYPE[2].Motion.Gluing_Nozzle_Z.Position[8].Pos := 0.0;
   PRODUCT_TYPE[2].Motion.Gluing_Nozzle_Z.Position[8].Vel := 200;
   PRODUCT_TYPE[3].Motion.Gluing_Nozzle_Z.Position[8].Pos := 0.0;
   PRODUCT_TYPE[3].Motion.Gluing_Nozzle_Z.Position[8].Vel := 200;
   PRODUCT_TYPE[4].Motion.Gluing_Nozzle_Z.Position[8].Pos := 0.0;
   PRODUCT_TYPE[4].Motion.Gluing_Nozzle_Z.Position[8].Vel := 200;
   PRODUCT_TYPE[5].Motion.Gluing_Nozzle_Z.Position[8].Pos := 0.0;
   PRODUCT_TYPE[5].Motion.Gluing_Nozzle_Z.Position[8].Vel := 200;
   PRODUCT_TYPE[6].Motion.Gluing_Nozzle_Z.Position[8].Pos := 0.0;
   PRODUCT_TYPE[6].Motion.Gluing_Nozzle_Z.Position[8].Vel := 200;
   PRODUCT_TYPE[7].Motion.Gluing_Nozzle_Z.Position[8].Pos := 0.0;
   PRODUCT_TYPE[7].Motion.Gluing_Nozzle_Z.Position[8].Vel := 200;
   PRODUCT_TYPE[8].Motion.Gluing_Nozzle_Z.Position[8].Pos := 0.0;
   PRODUCT_TYPE[8].Motion.Gluing_Nozzle_Z.Position[8].Vel := 200;
   PRODUCT_TYPE[9].Motion.Gluing_Nozzle_Z.Position[8].Pos := 0.0;
   PRODUCT_TYPE[9].Motion.Gluing_Nozzle_Z.Position[8].Vel := 200;
   PRODUCT_TYPE[10].Motion.Gluing_Nozzle_Z.Position[8].Pos := 0.0;
   PRODUCT_TYPE[10].Motion.Gluing_Nozzle_Z.Position[8].Vel := 200;
   PRODUCT_TYPE[1].Motion.Gluing_Nozzle_Z.Position[9].Pos := 123.0;
   PRODUCT_TYPE[1].Motion.Gluing_Nozzle_Z.Position[9].Vel := 200;
   PRODUCT_TYPE[2].Motion.Gluing_Nozzle_Z.Position[9].Pos := 123.0;
   PRODUCT_TYPE[2].Motion.Gluing_Nozzle_Z.Position[9].Vel := 200;
   PRODUCT_TYPE[3].Motion.Gluing_Nozzle_Z.Position[9].Pos := 123.0;
   PRODUCT_TYPE[3].Motion.Gluing_Nozzle_Z.Position[9].Vel := 200;
   PRODUCT_TYPE[4].Motion.Gluing_Nozzle_Z.Position[9].Pos := 123.0;
   PRODUCT_TYPE[4].Motion.Gluing_Nozzle_Z.Position[9].Vel := 200;
   PRODUCT_TYPE[5].Motion.Gluing_Nozzle_Z.Position[9].Pos := 123.0;
   PRODUCT_TYPE[5].Motion.Gluing_Nozzle_Z.Position[9].Vel := 200;
   PRODUCT_TYPE[6].Motion.Gluing_Nozzle_Z.Position[9].Pos := 123.0;
   PRODUCT_TYPE[6].Motion.Gluing_Nozzle_Z.Position[9].Vel := 200;
   PRODUCT_TYPE[7].Motion.Gluing_Nozzle_Z.Position[9].Pos := 123.0;
   PRODUCT_TYPE[7].Motion.Gluing_Nozzle_Z.Position[9].Vel := 200;
   PRODUCT_TYPE[8].Motion.Gluing_Nozzle_Z.Position[9].Pos := 123.0;
   PRODUCT_TYPE[8].Motion.Gluing_Nozzle_Z.Position[9].Vel := 200;
   PRODUCT_TYPE[9].Motion.Gluing_Nozzle_Z.Position[9].Pos := 123.0;
   PRODUCT_TYPE[9].Motion.Gluing_Nozzle_Z.Position[9].Vel := 200;
   PRODUCT_TYPE[10].Motion.Gluing_Nozzle_Z.Position[9].Pos := 123.0;
   PRODUCT_TYPE[10].Motion.Gluing_Nozzle_Z.Position[9].Vel := 200;
   PRODUCT_TYPE[1].Motion.Gluing_Nozzle_Z.Position[10].Pos := 0.0;
   PRODUCT_TYPE[1].Motion.Gluing_Nozzle_Z.Position[10].Vel := 0;
   PRODUCT_TYPE[2].Motion.Gluing_Nozzle_Z.Position[10].Pos := 0.0;
   PRODUCT_TYPE[2].Motion.Gluing_Nozzle_Z.Position[10].Vel := 0;
   PRODUCT_TYPE[3].Motion.Gluing_Nozzle_Z.Position[10].Pos := 0.0;
   PRODUCT_TYPE[3].Motion.Gluing_Nozzle_Z.Position[10].Vel := 0;
   PRODUCT_TYPE[4].Motion.Gluing_Nozzle_Z.Position[10].Pos := 0.0;
   PRODUCT_TYPE[4].Motion.Gluing_Nozzle_Z.Position[10].Vel := 0;
   PRODUCT_TYPE[5].Motion.Gluing_Nozzle_Z.Position[10].Pos := 0.0;
   PRODUCT_TYPE[5].Motion.Gluing_Nozzle_Z.Position[10].Vel := 0;
   PRODUCT_TYPE[6].Motion.Gluing_Nozzle_Z.Position[10].Pos := 0.0;
   PRODUCT_TYPE[6].Motion.Gluing_Nozzle_Z.Position[10].Vel := 0;
   PRODUCT_TYPE[7].Motion.Gluing_Nozzle_Z.Position[10].Pos := 0.0;
   PRODUCT_TYPE[7].Motion.Gluing_Nozzle_Z.Position[10].Vel := 0;
   PRODUCT_TYPE[8].Motion.Gluing_Nozzle_Z.Position[10].Pos := 0.0;
   PRODUCT_TYPE[8].Motion.Gluing_Nozzle_Z.Position[10].Vel := 0;
   PRODUCT_TYPE[9].Motion.Gluing_Nozzle_Z.Position[10].Pos := 0.0;
   PRODUCT_TYPE[9].Motion.Gluing_Nozzle_Z.Position[10].Vel := 0;
   PRODUCT_TYPE[10].Motion.Gluing_Nozzle_Z.Position[10].Pos := 0.0;
   PRODUCT_TYPE[10].Motion.Gluing_Nozzle_Z.Position[10].Vel := 0;
   PRODUCT_TYPE[1].Motion.Gluing_Nozzle_Z.Position[11].Pos := 0.0;
   PRODUCT_TYPE[1].Motion.Gluing_Nozzle_Z.Position[11].Vel := 0;
   PRODUCT_TYPE[2].Motion.Gluing_Nozzle_Z.Position[11].Pos := 0.0;
   PRODUCT_TYPE[2].Motion.Gluing_Nozzle_Z.Position[11].Vel := 0;
   PRODUCT_TYPE[3].Motion.Gluing_Nozzle_Z.Position[11].Pos := 0.0;
   PRODUCT_TYPE[3].Motion.Gluing_Nozzle_Z.Position[11].Vel := 0;
   PRODUCT_TYPE[4].Motion.Gluing_Nozzle_Z.Position[11].Pos := 0.0;
   PRODUCT_TYPE[4].Motion.Gluing_Nozzle_Z.Position[11].Vel := 0;
   PRODUCT_TYPE[5].Motion.Gluing_Nozzle_Z.Position[11].Pos := 0.0;
   PRODUCT_TYPE[5].Motion.Gluing_Nozzle_Z.Position[11].Vel := 0;
   PRODUCT_TYPE[6].Motion.Gluing_Nozzle_Z.Position[11].Pos := 0.0;
   PRODUCT_TYPE[6].Motion.Gluing_Nozzle_Z.Position[11].Vel := 0;
   PRODUCT_TYPE[7].Motion.Gluing_Nozzle_Z.Position[11].Pos := 0.0;
   PRODUCT_TYPE[7].Motion.Gluing_Nozzle_Z.Position[11].Vel := 0;
   PRODUCT_TYPE[8].Motion.Gluing_Nozzle_Z.Position[11].Pos := 0.0;
   PRODUCT_TYPE[8].Motion.Gluing_Nozzle_Z.Position[11].Vel := 0;
   PRODUCT_TYPE[9].Motion.Gluing_Nozzle_Z.Position[11].Pos := 0.0;
   PRODUCT_TYPE[9].Motion.Gluing_Nozzle_Z.Position[11].Vel := 0;
   PRODUCT_TYPE[10].Motion.Gluing_Nozzle_Z.Position[11].Pos := 0.0;
   PRODUCT_TYPE[10].Motion.Gluing_Nozzle_Z.Position[11].Vel := 0;
   PRODUCT_TYPE[1].Motion.Gluing_Nozzle_Z.Position[12].Pos := 0.0;
   PRODUCT_TYPE[1].Motion.Gluing_Nozzle_Z.Position[12].Vel := 0;
   PRODUCT_TYPE[2].Motion.Gluing_Nozzle_Z.Position[12].Pos := 0.0;
   PRODUCT_TYPE[2].Motion.Gluing_Nozzle_Z.Position[12].Vel := 0;
   PRODUCT_TYPE[3].Motion.Gluing_Nozzle_Z.Position[12].Pos := 0.0;
   PRODUCT_TYPE[3].Motion.Gluing_Nozzle_Z.Position[12].Vel := 0;
   PRODUCT_TYPE[4].Motion.Gluing_Nozzle_Z.Position[12].Pos := 0.0;
   PRODUCT_TYPE[4].Motion.Gluing_Nozzle_Z.Position[12].Vel := 0;
   PRODUCT_TYPE[5].Motion.Gluing_Nozzle_Z.Position[12].Pos := 0.0;
   PRODUCT_TYPE[5].Motion.Gluing_Nozzle_Z.Position[12].Vel := 0;
   PRODUCT_TYPE[6].Motion.Gluing_Nozzle_Z.Position[12].Pos := 0.0;
   PRODUCT_TYPE[6].Motion.Gluing_Nozzle_Z.Position[12].Vel := 0;
   PRODUCT_TYPE[7].Motion.Gluing_Nozzle_Z.Position[12].Pos := 0.0;
   PRODUCT_TYPE[7].Motion.Gluing_Nozzle_Z.Position[12].Vel := 0;
   PRODUCT_TYPE[8].Motion.Gluing_Nozzle_Z.Position[12].Pos := 0.0;
   PRODUCT_TYPE[8].Motion.Gluing_Nozzle_Z.Position[12].Vel := 0;
   PRODUCT_TYPE[9].Motion.Gluing_Nozzle_Z.Position[12].Pos := 0.0;
   PRODUCT_TYPE[9].Motion.Gluing_Nozzle_Z.Position[12].Vel := 0;
   PRODUCT_TYPE[10].Motion.Gluing_Nozzle_Z.Position[12].Pos := 0.0;
   PRODUCT_TYPE[10].Motion.Gluing_Nozzle_Z.Position[12].Vel := 0;
   PRODUCT_TYPE[1].Motion.Gluing_Nozzle_Z.Position[13].Pos := 0.0;
   PRODUCT_TYPE[1].Motion.Gluing_Nozzle_Z.Position[13].Vel := 0;
   PRODUCT_TYPE[2].Motion.Gluing_Nozzle_Z.Position[13].Pos := 0.0;
   PRODUCT_TYPE[2].Motion.Gluing_Nozzle_Z.Position[13].Vel := 0;
   PRODUCT_TYPE[3].Motion.Gluing_Nozzle_Z.Position[13].Pos := 0.0;
   PRODUCT_TYPE[3].Motion.Gluing_Nozzle_Z.Position[13].Vel := 0;
   PRODUCT_TYPE[4].Motion.Gluing_Nozzle_Z.Position[13].Pos := 0.0;
   PRODUCT_TYPE[4].Motion.Gluing_Nozzle_Z.Position[13].Vel := 0;
   PRODUCT_TYPE[5].Motion.Gluing_Nozzle_Z.Position[13].Pos := 0.0;
   PRODUCT_TYPE[5].Motion.Gluing_Nozzle_Z.Position[13].Vel := 0;
   PRODUCT_TYPE[6].Motion.Gluing_Nozzle_Z.Position[13].Pos := 0.0;
   PRODUCT_TYPE[6].Motion.Gluing_Nozzle_Z.Position[13].Vel := 0;
   PRODUCT_TYPE[7].Motion.Gluing_Nozzle_Z.Position[13].Pos := 0.0;
   PRODUCT_TYPE[7].Motion.Gluing_Nozzle_Z.Position[13].Vel := 0;
   PRODUCT_TYPE[8].Motion.Gluing_Nozzle_Z.Position[13].Pos := 0.0;
   PRODUCT_TYPE[8].Motion.Gluing_Nozzle_Z.Position[13].Vel := 0;
   PRODUCT_TYPE[9].Motion.Gluing_Nozzle_Z.Position[13].Pos := 0.0;
   PRODUCT_TYPE[9].Motion.Gluing_Nozzle_Z.Position[13].Vel := 0;
   PRODUCT_TYPE[10].Motion.Gluing_Nozzle_Z.Position[13].Pos := 0.0;
   PRODUCT_TYPE[10].Motion.Gluing_Nozzle_Z.Position[13].Vel := 0;
   PRODUCT_TYPE[1].Motion.Gluing_Nozzle_Z.Position[14].Pos := 0.0;
   PRODUCT_TYPE[1].Motion.Gluing_Nozzle_Z.Position[14].Vel := 0;
   PRODUCT_TYPE[2].Motion.Gluing_Nozzle_Z.Position[14].Pos := 0.0;
   PRODUCT_TYPE[2].Motion.Gluing_Nozzle_Z.Position[14].Vel := 0;
   PRODUCT_TYPE[3].Motion.Gluing_Nozzle_Z.Position[14].Pos := 0.0;
   PRODUCT_TYPE[3].Motion.Gluing_Nozzle_Z.Position[14].Vel := 0;
   PRODUCT_TYPE[4].Motion.Gluing_Nozzle_Z.Position[14].Pos := 0.0;
   PRODUCT_TYPE[4].Motion.Gluing_Nozzle_Z.Position[14].Vel := 0;
   PRODUCT_TYPE[5].Motion.Gluing_Nozzle_Z.Position[14].Pos := 0.0;
   PRODUCT_TYPE[5].Motion.Gluing_Nozzle_Z.Position[14].Vel := 0;
   PRODUCT_TYPE[6].Motion.Gluing_Nozzle_Z.Position[14].Pos := 0.0;
   PRODUCT_TYPE[6].Motion.Gluing_Nozzle_Z.Position[14].Vel := 0;
   PRODUCT_TYPE[7].Motion.Gluing_Nozzle_Z.Position[14].Pos := 0.0;
   PRODUCT_TYPE[7].Motion.Gluing_Nozzle_Z.Position[14].Vel := 0;
   PRODUCT_TYPE[8].Motion.Gluing_Nozzle_Z.Position[14].Pos := 0.0;
   PRODUCT_TYPE[8].Motion.Gluing_Nozzle_Z.Position[14].Vel := 0;
   PRODUCT_TYPE[9].Motion.Gluing_Nozzle_Z.Position[14].Pos := 0.0;
   PRODUCT_TYPE[9].Motion.Gluing_Nozzle_Z.Position[14].Vel := 0;
   PRODUCT_TYPE[10].Motion.Gluing_Nozzle_Z.Position[14].Pos := 0.0;
   PRODUCT_TYPE[10].Motion.Gluing_Nozzle_Z.Position[14].Vel := 0;
   PRODUCT_TYPE[1].Motion.Gluing_Nozzle_Z.Position[15].Pos := 0.0;
   PRODUCT_TYPE[1].Motion.Gluing_Nozzle_Z.Position[15].Vel := 0;
   PRODUCT_TYPE[2].Motion.Gluing_Nozzle_Z.Position[15].Pos := 0.0;
   PRODUCT_TYPE[2].Motion.Gluing_Nozzle_Z.Position[15].Vel := 0;
   PRODUCT_TYPE[3].Motion.Gluing_Nozzle_Z.Position[15].Pos := 0.0;
   PRODUCT_TYPE[3].Motion.Gluing_Nozzle_Z.Position[15].Vel := 0;
   PRODUCT_TYPE[4].Motion.Gluing_Nozzle_Z.Position[15].Pos := 0.0;
   PRODUCT_TYPE[4].Motion.Gluing_Nozzle_Z.Position[15].Vel := 0;
   PRODUCT_TYPE[5].Motion.Gluing_Nozzle_Z.Position[15].Pos := 0.0;
   PRODUCT_TYPE[5].Motion.Gluing_Nozzle_Z.Position[15].Vel := 0;
   PRODUCT_TYPE[6].Motion.Gluing_Nozzle_Z.Position[15].Pos := 0.0;
   PRODUCT_TYPE[6].Motion.Gluing_Nozzle_Z.Position[15].Vel := 0;
   PRODUCT_TYPE[7].Motion.Gluing_Nozzle_Z.Position[15].Pos := 0.0;
   PRODUCT_TYPE[7].Motion.Gluing_Nozzle_Z.Position[15].Vel := 0;
   PRODUCT_TYPE[8].Motion.Gluing_Nozzle_Z.Position[15].Pos := 0.0;
   PRODUCT_TYPE[8].Motion.Gluing_Nozzle_Z.Position[15].Vel := 0;
   PRODUCT_TYPE[9].Motion.Gluing_Nozzle_Z.Position[15].Pos := 0.0;
   PRODUCT_TYPE[9].Motion.Gluing_Nozzle_Z.Position[15].Vel := 0;
   PRODUCT_TYPE[10].Motion.Gluing_Nozzle_Z.Position[15].Pos := 0.0;
   PRODUCT_TYPE[10].Motion.Gluing_Nozzle_Z.Position[15].Vel := 0;
   PRODUCT_TYPE[1].Motion.Gluing_Nozzle_Z.Position[16].Pos := 0.0;
   PRODUCT_TYPE[1].Motion.Gluing_Nozzle_Z.Position[16].Vel := 0;
   PRODUCT_TYPE[2].Motion.Gluing_Nozzle_Z.Position[16].Pos := 0.0;
   PRODUCT_TYPE[2].Motion.Gluing_Nozzle_Z.Position[16].Vel := 0;
   PRODUCT_TYPE[3].Motion.Gluing_Nozzle_Z.Position[16].Pos := 0.0;
   PRODUCT_TYPE[3].Motion.Gluing_Nozzle_Z.Position[16].Vel := 0;
   PRODUCT_TYPE[4].Motion.Gluing_Nozzle_Z.Position[16].Pos := 0.0;
   PRODUCT_TYPE[4].Motion.Gluing_Nozzle_Z.Position[16].Vel := 0;
   PRODUCT_TYPE[5].Motion.Gluing_Nozzle_Z.Position[16].Pos := 0.0;
   PRODUCT_TYPE[5].Motion.Gluing_Nozzle_Z.Position[16].Vel := 0;
   PRODUCT_TYPE[6].Motion.Gluing_Nozzle_Z.Position[16].Pos := 0.0;
   PRODUCT_TYPE[6].Motion.Gluing_Nozzle_Z.Position[16].Vel := 0;
   PRODUCT_TYPE[7].Motion.Gluing_Nozzle_Z.Position[16].Pos := 0.0;
   PRODUCT_TYPE[7].Motion.Gluing_Nozzle_Z.Position[16].Vel := 0;
   PRODUCT_TYPE[8].Motion.Gluing_Nozzle_Z.Position[16].Pos := 0.0;
   PRODUCT_TYPE[8].Motion.Gluing_Nozzle_Z.Position[16].Vel := 0;
   PRODUCT_TYPE[9].Motion.Gluing_Nozzle_Z.Position[16].Pos := 0.0;
   PRODUCT_TYPE[9].Motion.Gluing_Nozzle_Z.Position[16].Vel := 0;
   PRODUCT_TYPE[10].Motion.Gluing_Nozzle_Z.Position[16].Pos := 0.0;
   PRODUCT_TYPE[10].Motion.Gluing_Nozzle_Z.Position[16].Vel := 0;
   PRODUCT_TYPE[1].Motion.Gluing_Nozzle_Z.Position[17].Pos := 0.0;
   PRODUCT_TYPE[1].Motion.Gluing_Nozzle_Z.Position[17].Vel := 0;
   PRODUCT_TYPE[2].Motion.Gluing_Nozzle_Z.Position[17].Pos := 0.0;
   PRODUCT_TYPE[2].Motion.Gluing_Nozzle_Z.Position[17].Vel := 0;
   PRODUCT_TYPE[3].Motion.Gluing_Nozzle_Z.Position[17].Pos := 0.0;
   PRODUCT_TYPE[3].Motion.Gluing_Nozzle_Z.Position[17].Vel := 0;
   PRODUCT_TYPE[4].Motion.Gluing_Nozzle_Z.Position[17].Pos := 0.0;
   PRODUCT_TYPE[4].Motion.Gluing_Nozzle_Z.Position[17].Vel := 0;
   PRODUCT_TYPE[5].Motion.Gluing_Nozzle_Z.Position[17].Pos := 0.0;
   PRODUCT_TYPE[5].Motion.Gluing_Nozzle_Z.Position[17].Vel := 0;
   PRODUCT_TYPE[6].Motion.Gluing_Nozzle_Z.Position[17].Pos := 0.0;
   PRODUCT_TYPE[6].Motion.Gluing_Nozzle_Z.Position[17].Vel := 0;
   PRODUCT_TYPE[7].Motion.Gluing_Nozzle_Z.Position[17].Pos := 0.0;
   PRODUCT_TYPE[7].Motion.Gluing_Nozzle_Z.Position[17].Vel := 0;
   PRODUCT_TYPE[8].Motion.Gluing_Nozzle_Z.Position[17].Pos := 0.0;
   PRODUCT_TYPE[8].Motion.Gluing_Nozzle_Z.Position[17].Vel := 0;
   PRODUCT_TYPE[9].Motion.Gluing_Nozzle_Z.Position[17].Pos := 0.0;
   PRODUCT_TYPE[9].Motion.Gluing_Nozzle_Z.Position[17].Vel := 0;
   PRODUCT_TYPE[10].Motion.Gluing_Nozzle_Z.Position[17].Pos := 0.0;
   PRODUCT_TYPE[10].Motion.Gluing_Nozzle_Z.Position[17].Vel := 0;
   PRODUCT_TYPE[1].Motion.Gluing_Nozzle_Z.Position[18].Pos := 0.0;
   PRODUCT_TYPE[1].Motion.Gluing_Nozzle_Z.Position[18].Vel := 0;
   PRODUCT_TYPE[2].Motion.Gluing_Nozzle_Z.Position[18].Pos := 0.0;
   PRODUCT_TYPE[2].Motion.Gluing_Nozzle_Z.Position[18].Vel := 0;
   PRODUCT_TYPE[3].Motion.Gluing_Nozzle_Z.Position[18].Pos := 0.0;
   PRODUCT_TYPE[3].Motion.Gluing_Nozzle_Z.Position[18].Vel := 0;
   PRODUCT_TYPE[4].Motion.Gluing_Nozzle_Z.Position[18].Pos := 0.0;
   PRODUCT_TYPE[4].Motion.Gluing_Nozzle_Z.Position[18].Vel := 0;
   PRODUCT_TYPE[5].Motion.Gluing_Nozzle_Z.Position[18].Pos := 0.0;
   PRODUCT_TYPE[5].Motion.Gluing_Nozzle_Z.Position[18].Vel := 0;
   PRODUCT_TYPE[6].Motion.Gluing_Nozzle_Z.Position[18].Pos := 0.0;
   PRODUCT_TYPE[6].Motion.Gluing_Nozzle_Z.Position[18].Vel := 0;
   PRODUCT_TYPE[7].Motion.Gluing_Nozzle_Z.Position[18].Pos := 0.0;
   PRODUCT_TYPE[7].Motion.Gluing_Nozzle_Z.Position[18].Vel := 0;
   PRODUCT_TYPE[8].Motion.Gluing_Nozzle_Z.Position[18].Pos := 0.0;
   PRODUCT_TYPE[8].Motion.Gluing_Nozzle_Z.Position[18].Vel := 0;
   PRODUCT_TYPE[9].Motion.Gluing_Nozzle_Z.Position[18].Pos := 0.0;
   PRODUCT_TYPE[9].Motion.Gluing_Nozzle_Z.Position[18].Vel := 0;
   PRODUCT_TYPE[10].Motion.Gluing_Nozzle_Z.Position[18].Pos := 0.0;
   PRODUCT_TYPE[10].Motion.Gluing_Nozzle_Z.Position[18].Vel := 0;
   PRODUCT_TYPE[1].Motion.Gluing_Nozzle_Z.Position[19].Pos := 0.0;
   PRODUCT_TYPE[1].Motion.Gluing_Nozzle_Z.Position[19].Vel := 0;
   PRODUCT_TYPE[2].Motion.Gluing_Nozzle_Z.Position[19].Pos := 0.0;
   PRODUCT_TYPE[2].Motion.Gluing_Nozzle_Z.Position[19].Vel := 0;
   PRODUCT_TYPE[3].Motion.Gluing_Nozzle_Z.Position[19].Pos := 0.0;
   PRODUCT_TYPE[3].Motion.Gluing_Nozzle_Z.Position[19].Vel := 0;
   PRODUCT_TYPE[4].Motion.Gluing_Nozzle_Z.Position[19].Pos := 0.0;
   PRODUCT_TYPE[4].Motion.Gluing_Nozzle_Z.Position[19].Vel := 0;
   PRODUCT_TYPE[5].Motion.Gluing_Nozzle_Z.Position[19].Pos := 0.0;
   PRODUCT_TYPE[5].Motion.Gluing_Nozzle_Z.Position[19].Vel := 0;
   PRODUCT_TYPE[6].Motion.Gluing_Nozzle_Z.Position[19].Pos := 0.0;
   PRODUCT_TYPE[6].Motion.Gluing_Nozzle_Z.Position[19].Vel := 0;
   PRODUCT_TYPE[7].Motion.Gluing_Nozzle_Z.Position[19].Pos := 0.0;
   PRODUCT_TYPE[7].Motion.Gluing_Nozzle_Z.Position[19].Vel := 0;
   PRODUCT_TYPE[8].Motion.Gluing_Nozzle_Z.Position[19].Pos := 0.0;
   PRODUCT_TYPE[8].Motion.Gluing_Nozzle_Z.Position[19].Vel := 0;
   PRODUCT_TYPE[9].Motion.Gluing_Nozzle_Z.Position[19].Pos := 0.0;
   PRODUCT_TYPE[9].Motion.Gluing_Nozzle_Z.Position[19].Vel := 0;
   PRODUCT_TYPE[10].Motion.Gluing_Nozzle_Z.Position[19].Pos := 0.0;
   PRODUCT_TYPE[10].Motion.Gluing_Nozzle_Z.Position[19].Vel := 0;
   PRODUCT_TYPE[1].Motion.Gluing_Nozzle_Z.Position[20].Pos := 0.0;
   PRODUCT_TYPE[1].Motion.Gluing_Nozzle_Z.Position[20].Vel := 0;
   PRODUCT_TYPE[2].Motion.Gluing_Nozzle_Z.Position[20].Pos := 0.0;
   PRODUCT_TYPE[2].Motion.Gluing_Nozzle_Z.Position[20].Vel := 0;
   PRODUCT_TYPE[3].Motion.Gluing_Nozzle_Z.Position[20].Pos := 0.0;
   PRODUCT_TYPE[3].Motion.Gluing_Nozzle_Z.Position[20].Vel := 0;
   PRODUCT_TYPE[4].Motion.Gluing_Nozzle_Z.Position[20].Pos := 0.0;
   PRODUCT_TYPE[4].Motion.Gluing_Nozzle_Z.Position[20].Vel := 0;
   PRODUCT_TYPE[5].Motion.Gluing_Nozzle_Z.Position[20].Pos := 0.0;
   PRODUCT_TYPE[5].Motion.Gluing_Nozzle_Z.Position[20].Vel := 0;
   PRODUCT_TYPE[6].Motion.Gluing_Nozzle_Z.Position[20].Pos := 0.0;
   PRODUCT_TYPE[6].Motion.Gluing_Nozzle_Z.Position[20].Vel := 0;
   PRODUCT_TYPE[7].Motion.Gluing_Nozzle_Z.Position[20].Pos := 0.0;
   PRODUCT_TYPE[7].Motion.Gluing_Nozzle_Z.Position[20].Vel := 0;
   PRODUCT_TYPE[8].Motion.Gluing_Nozzle_Z.Position[20].Pos := 0.0;
   PRODUCT_TYPE[8].Motion.Gluing_Nozzle_Z.Position[20].Vel := 0;
   PRODUCT_TYPE[9].Motion.Gluing_Nozzle_Z.Position[20].Pos := 0.0;
   PRODUCT_TYPE[9].Motion.Gluing_Nozzle_Z.Position[20].Vel := 0;
   PRODUCT_TYPE[10].Motion.Gluing_Nozzle_Z.Position[20].Pos := 0.0;
   PRODUCT_TYPE[10].Motion.Gluing_Nozzle_Z.Position[20].Vel := 0;
   PRODUCT_TYPE[1].Motion.Gluing_Nozzle_X.Position[1].Pos := 2.34;
   PRODUCT_TYPE[1].Motion.Gluing_Nozzle_X.Position[1].Vel := 200;
   PRODUCT_TYPE[2].Motion.Gluing_Nozzle_X.Position[1].Pos := 2.34;
   PRODUCT_TYPE[2].Motion.Gluing_Nozzle_X.Position[1].Vel := 200;
   PRODUCT_TYPE[3].Motion.Gluing_Nozzle_X.Position[1].Pos := 2.34;
   PRODUCT_TYPE[3].Motion.Gluing_Nozzle_X.Position[1].Vel := 200;
   PRODUCT_TYPE[4].Motion.Gluing_Nozzle_X.Position[1].Pos := 2.34;
   PRODUCT_TYPE[4].Motion.Gluing_Nozzle_X.Position[1].Vel := 200;
   PRODUCT_TYPE[5].Motion.Gluing_Nozzle_X.Position[1].Pos := 2.34;
   PRODUCT_TYPE[5].Motion.Gluing_Nozzle_X.Position[1].Vel := 200;
   PRODUCT_TYPE[6].Motion.Gluing_Nozzle_X.Position[1].Pos := 2.34;
   PRODUCT_TYPE[6].Motion.Gluing_Nozzle_X.Position[1].Vel := 200;
   PRODUCT_TYPE[7].Motion.Gluing_Nozzle_X.Position[1].Pos := 2.34;
   PRODUCT_TYPE[7].Motion.Gluing_Nozzle_X.Position[1].Vel := 200;
   PRODUCT_TYPE[8].Motion.Gluing_Nozzle_X.Position[1].Pos := 2.34;
   PRODUCT_TYPE[8].Motion.Gluing_Nozzle_X.Position[1].Vel := 200;
   PRODUCT_TYPE[9].Motion.Gluing_Nozzle_X.Position[1].Pos := 2.34;
   PRODUCT_TYPE[9].Motion.Gluing_Nozzle_X.Position[1].Vel := 200;
   PRODUCT_TYPE[10].Motion.Gluing_Nozzle_X.Position[1].Pos := 2.34;
   PRODUCT_TYPE[10].Motion.Gluing_Nozzle_X.Position[1].Vel := 200;
   PRODUCT_TYPE[1].Motion.Gluing_Nozzle_X.Position[2].Pos := 76.0;
   PRODUCT_TYPE[1].Motion.Gluing_Nozzle_X.Position[2].Vel := 200;
   PRODUCT_TYPE[2].Motion.Gluing_Nozzle_X.Position[2].Pos := 76.0;
   PRODUCT_TYPE[2].Motion.Gluing_Nozzle_X.Position[2].Vel := 200;
   PRODUCT_TYPE[3].Motion.Gluing_Nozzle_X.Position[2].Pos := 76.0;
   PRODUCT_TYPE[3].Motion.Gluing_Nozzle_X.Position[2].Vel := 200;
   PRODUCT_TYPE[4].Motion.Gluing_Nozzle_X.Position[2].Pos := 76.0;
   PRODUCT_TYPE[4].Motion.Gluing_Nozzle_X.Position[2].Vel := 200;
   PRODUCT_TYPE[5].Motion.Gluing_Nozzle_X.Position[2].Pos := 76.0;
   PRODUCT_TYPE[5].Motion.Gluing_Nozzle_X.Position[2].Vel := 200;
   PRODUCT_TYPE[6].Motion.Gluing_Nozzle_X.Position[2].Pos := 76.0;
   PRODUCT_TYPE[6].Motion.Gluing_Nozzle_X.Position[2].Vel := 200;
   PRODUCT_TYPE[7].Motion.Gluing_Nozzle_X.Position[2].Pos := 76.0;
   PRODUCT_TYPE[7].Motion.Gluing_Nozzle_X.Position[2].Vel := 200;
   PRODUCT_TYPE[8].Motion.Gluing_Nozzle_X.Position[2].Pos := 76.0;
   PRODUCT_TYPE[8].Motion.Gluing_Nozzle_X.Position[2].Vel := 200;
   PRODUCT_TYPE[9].Motion.Gluing_Nozzle_X.Position[2].Pos := 76.0;
   PRODUCT_TYPE[9].Motion.Gluing_Nozzle_X.Position[2].Vel := 200;
   PRODUCT_TYPE[10].Motion.Gluing_Nozzle_X.Position[2].Pos := 76.0;
   PRODUCT_TYPE[10].Motion.Gluing_Nozzle_X.Position[2].Vel := 200;
   PRODUCT_TYPE[1].Motion.Gluing_Nozzle_X.Position[3].Pos := 84.69;
   PRODUCT_TYPE[1].Motion.Gluing_Nozzle_X.Position[3].Vel := 200;
   PRODUCT_TYPE[2].Motion.Gluing_Nozzle_X.Position[3].Pos := 84.69;
   PRODUCT_TYPE[2].Motion.Gluing_Nozzle_X.Position[3].Vel := 200;
   PRODUCT_TYPE[3].Motion.Gluing_Nozzle_X.Position[3].Pos := 84.69;
   PRODUCT_TYPE[3].Motion.Gluing_Nozzle_X.Position[3].Vel := 200;
   PRODUCT_TYPE[4].Motion.Gluing_Nozzle_X.Position[3].Pos := 84.69;
   PRODUCT_TYPE[4].Motion.Gluing_Nozzle_X.Position[3].Vel := 200;
   PRODUCT_TYPE[5].Motion.Gluing_Nozzle_X.Position[3].Pos := 84.69;
   PRODUCT_TYPE[5].Motion.Gluing_Nozzle_X.Position[3].Vel := 200;
   PRODUCT_TYPE[6].Motion.Gluing_Nozzle_X.Position[3].Pos := 84.69;
   PRODUCT_TYPE[6].Motion.Gluing_Nozzle_X.Position[3].Vel := 200;
   PRODUCT_TYPE[7].Motion.Gluing_Nozzle_X.Position[3].Pos := 84.69;
   PRODUCT_TYPE[7].Motion.Gluing_Nozzle_X.Position[3].Vel := 200;
   PRODUCT_TYPE[8].Motion.Gluing_Nozzle_X.Position[3].Pos := 84.69;
   PRODUCT_TYPE[8].Motion.Gluing_Nozzle_X.Position[3].Vel := 200;
   PRODUCT_TYPE[9].Motion.Gluing_Nozzle_X.Position[3].Pos := 84.69;
   PRODUCT_TYPE[9].Motion.Gluing_Nozzle_X.Position[3].Vel := 200;
   PRODUCT_TYPE[10].Motion.Gluing_Nozzle_X.Position[3].Pos := 84.69;
   PRODUCT_TYPE[10].Motion.Gluing_Nozzle_X.Position[3].Vel := 200;
   PRODUCT_TYPE[1].Motion.Gluing_Nozzle_X.Position[4].Pos := 84.69;
   PRODUCT_TYPE[1].Motion.Gluing_Nozzle_X.Position[4].Vel := 200;
   PRODUCT_TYPE[2].Motion.Gluing_Nozzle_X.Position[4].Pos := 84.69;
   PRODUCT_TYPE[2].Motion.Gluing_Nozzle_X.Position[4].Vel := 200;
   PRODUCT_TYPE[3].Motion.Gluing_Nozzle_X.Position[4].Pos := 84.69;
   PRODUCT_TYPE[3].Motion.Gluing_Nozzle_X.Position[4].Vel := 200;
   PRODUCT_TYPE[4].Motion.Gluing_Nozzle_X.Position[4].Pos := 84.69;
   PRODUCT_TYPE[4].Motion.Gluing_Nozzle_X.Position[4].Vel := 200;
   PRODUCT_TYPE[5].Motion.Gluing_Nozzle_X.Position[4].Pos := 84.69;
   PRODUCT_TYPE[5].Motion.Gluing_Nozzle_X.Position[4].Vel := 200;
   PRODUCT_TYPE[6].Motion.Gluing_Nozzle_X.Position[4].Pos := 84.69;
   PRODUCT_TYPE[6].Motion.Gluing_Nozzle_X.Position[4].Vel := 200;
   PRODUCT_TYPE[7].Motion.Gluing_Nozzle_X.Position[4].Pos := 84.69;
   PRODUCT_TYPE[7].Motion.Gluing_Nozzle_X.Position[4].Vel := 200;
   PRODUCT_TYPE[8].Motion.Gluing_Nozzle_X.Position[4].Pos := 84.69;
   PRODUCT_TYPE[8].Motion.Gluing_Nozzle_X.Position[4].Vel := 200;
   PRODUCT_TYPE[9].Motion.Gluing_Nozzle_X.Position[4].Pos := 84.69;
   PRODUCT_TYPE[9].Motion.Gluing_Nozzle_X.Position[4].Vel := 200;
   PRODUCT_TYPE[10].Motion.Gluing_Nozzle_X.Position[4].Pos := 84.69;
   PRODUCT_TYPE[10].Motion.Gluing_Nozzle_X.Position[4].Vel := 200;
   PRODUCT_TYPE[1].Motion.Gluing_Nozzle_X.Position[5].Pos := 84.69;
   PRODUCT_TYPE[1].Motion.Gluing_Nozzle_X.Position[5].Vel := 200;
   PRODUCT_TYPE[2].Motion.Gluing_Nozzle_X.Position[5].Pos := 84.69;
   PRODUCT_TYPE[2].Motion.Gluing_Nozzle_X.Position[5].Vel := 200;
   PRODUCT_TYPE[3].Motion.Gluing_Nozzle_X.Position[5].Pos := 84.69;
   PRODUCT_TYPE[3].Motion.Gluing_Nozzle_X.Position[5].Vel := 200;
   PRODUCT_TYPE[4].Motion.Gluing_Nozzle_X.Position[5].Pos := 84.69;
   PRODUCT_TYPE[4].Motion.Gluing_Nozzle_X.Position[5].Vel := 200;
   PRODUCT_TYPE[5].Motion.Gluing_Nozzle_X.Position[5].Pos := 84.69;
   PRODUCT_TYPE[5].Motion.Gluing_Nozzle_X.Position[5].Vel := 200;
   PRODUCT_TYPE[6].Motion.Gluing_Nozzle_X.Position[5].Pos := 84.69;
   PRODUCT_TYPE[6].Motion.Gluing_Nozzle_X.Position[5].Vel := 200;
   PRODUCT_TYPE[7].Motion.Gluing_Nozzle_X.Position[5].Pos := 84.69;
   PRODUCT_TYPE[7].Motion.Gluing_Nozzle_X.Position[5].Vel := 200;
   PRODUCT_TYPE[8].Motion.Gluing_Nozzle_X.Position[5].Pos := 84.69;
   PRODUCT_TYPE[8].Motion.Gluing_Nozzle_X.Position[5].Vel := 200;
   PRODUCT_TYPE[9].Motion.Gluing_Nozzle_X.Position[5].Pos := 84.69;
   PRODUCT_TYPE[9].Motion.Gluing_Nozzle_X.Position[5].Vel := 200;
   PRODUCT_TYPE[10].Motion.Gluing_Nozzle_X.Position[5].Pos := 84.69;
   PRODUCT_TYPE[10].Motion.Gluing_Nozzle_X.Position[5].Vel := 200;
   PRODUCT_TYPE[1].Motion.Gluing_Nozzle_X.Position[6].Pos := 84.69;
   PRODUCT_TYPE[1].Motion.Gluing_Nozzle_X.Position[6].Vel := 200;
   PRODUCT_TYPE[2].Motion.Gluing_Nozzle_X.Position[6].Pos := 84.69;
   PRODUCT_TYPE[2].Motion.Gluing_Nozzle_X.Position[6].Vel := 200;
   PRODUCT_TYPE[3].Motion.Gluing_Nozzle_X.Position[6].Pos := 84.69;
   PRODUCT_TYPE[3].Motion.Gluing_Nozzle_X.Position[6].Vel := 200;
   PRODUCT_TYPE[4].Motion.Gluing_Nozzle_X.Position[6].Pos := 84.69;
   PRODUCT_TYPE[4].Motion.Gluing_Nozzle_X.Position[6].Vel := 200;
   PRODUCT_TYPE[5].Motion.Gluing_Nozzle_X.Position[6].Pos := 84.69;
   PRODUCT_TYPE[5].Motion.Gluing_Nozzle_X.Position[6].Vel := 200;
   PRODUCT_TYPE[6].Motion.Gluing_Nozzle_X.Position[6].Pos := 84.69;
   PRODUCT_TYPE[6].Motion.Gluing_Nozzle_X.Position[6].Vel := 200;
   PRODUCT_TYPE[7].Motion.Gluing_Nozzle_X.Position[6].Pos := 84.69;
   PRODUCT_TYPE[7].Motion.Gluing_Nozzle_X.Position[6].Vel := 200;
   PRODUCT_TYPE[8].Motion.Gluing_Nozzle_X.Position[6].Pos := 84.69;
   PRODUCT_TYPE[8].Motion.Gluing_Nozzle_X.Position[6].Vel := 200;
   PRODUCT_TYPE[9].Motion.Gluing_Nozzle_X.Position[6].Pos := 84.69;
   PRODUCT_TYPE[9].Motion.Gluing_Nozzle_X.Position[6].Vel := 200;
   PRODUCT_TYPE[10].Motion.Gluing_Nozzle_X.Position[6].Pos := 84.69;
   PRODUCT_TYPE[10].Motion.Gluing_Nozzle_X.Position[6].Vel := 200;
   PRODUCT_TYPE[1].Motion.Gluing_Nozzle_X.Position[7].Pos := 85.0;
   PRODUCT_TYPE[1].Motion.Gluing_Nozzle_X.Position[7].Vel := 200;
   PRODUCT_TYPE[2].Motion.Gluing_Nozzle_X.Position[7].Pos := 85.0;
   PRODUCT_TYPE[2].Motion.Gluing_Nozzle_X.Position[7].Vel := 200;
   PRODUCT_TYPE[3].Motion.Gluing_Nozzle_X.Position[7].Pos := 85.0;
   PRODUCT_TYPE[3].Motion.Gluing_Nozzle_X.Position[7].Vel := 200;
   PRODUCT_TYPE[4].Motion.Gluing_Nozzle_X.Position[7].Pos := 85.0;
   PRODUCT_TYPE[4].Motion.Gluing_Nozzle_X.Position[7].Vel := 200;
   PRODUCT_TYPE[5].Motion.Gluing_Nozzle_X.Position[7].Pos := 85.0;
   PRODUCT_TYPE[5].Motion.Gluing_Nozzle_X.Position[7].Vel := 200;
   PRODUCT_TYPE[6].Motion.Gluing_Nozzle_X.Position[7].Pos := 85.0;
   PRODUCT_TYPE[6].Motion.Gluing_Nozzle_X.Position[7].Vel := 200;
   PRODUCT_TYPE[7].Motion.Gluing_Nozzle_X.Position[7].Pos := 85.0;
   PRODUCT_TYPE[7].Motion.Gluing_Nozzle_X.Position[7].Vel := 200;
   PRODUCT_TYPE[8].Motion.Gluing_Nozzle_X.Position[7].Pos := 85.0;
   PRODUCT_TYPE[8].Motion.Gluing_Nozzle_X.Position[7].Vel := 200;
   PRODUCT_TYPE[9].Motion.Gluing_Nozzle_X.Position[7].Pos := 85.0;
   PRODUCT_TYPE[9].Motion.Gluing_Nozzle_X.Position[7].Vel := 200;
   PRODUCT_TYPE[10].Motion.Gluing_Nozzle_X.Position[7].Pos := 85.0;
   PRODUCT_TYPE[10].Motion.Gluing_Nozzle_X.Position[7].Vel := 200;
   PRODUCT_TYPE[1].Motion.Gluing_Nozzle_X.Position[8].Pos := 88.53;
   PRODUCT_TYPE[1].Motion.Gluing_Nozzle_X.Position[8].Vel := 200;
   PRODUCT_TYPE[2].Motion.Gluing_Nozzle_X.Position[8].Pos := 88.53;
   PRODUCT_TYPE[2].Motion.Gluing_Nozzle_X.Position[8].Vel := 200;
   PRODUCT_TYPE[3].Motion.Gluing_Nozzle_X.Position[8].Pos := 88.53;
   PRODUCT_TYPE[3].Motion.Gluing_Nozzle_X.Position[8].Vel := 200;
   PRODUCT_TYPE[4].Motion.Gluing_Nozzle_X.Position[8].Pos := 88.53;
   PRODUCT_TYPE[4].Motion.Gluing_Nozzle_X.Position[8].Vel := 200;
   PRODUCT_TYPE[5].Motion.Gluing_Nozzle_X.Position[8].Pos := 88.53;
   PRODUCT_TYPE[5].Motion.Gluing_Nozzle_X.Position[8].Vel := 200;
   PRODUCT_TYPE[6].Motion.Gluing_Nozzle_X.Position[8].Pos := 88.53;
   PRODUCT_TYPE[6].Motion.Gluing_Nozzle_X.Position[8].Vel := 200;
   PRODUCT_TYPE[7].Motion.Gluing_Nozzle_X.Position[8].Pos := 88.53;
   PRODUCT_TYPE[7].Motion.Gluing_Nozzle_X.Position[8].Vel := 200;
   PRODUCT_TYPE[8].Motion.Gluing_Nozzle_X.Position[8].Pos := 88.53;
   PRODUCT_TYPE[8].Motion.Gluing_Nozzle_X.Position[8].Vel := 200;
   PRODUCT_TYPE[9].Motion.Gluing_Nozzle_X.Position[8].Pos := 88.53;
   PRODUCT_TYPE[9].Motion.Gluing_Nozzle_X.Position[8].Vel := 200;
   PRODUCT_TYPE[10].Motion.Gluing_Nozzle_X.Position[8].Pos := 88.53;
   PRODUCT_TYPE[10].Motion.Gluing_Nozzle_X.Position[8].Vel := 200;
   PRODUCT_TYPE[1].Motion.Gluing_Nozzle_X.Position[9].Pos := 0.0;
   PRODUCT_TYPE[1].Motion.Gluing_Nozzle_X.Position[9].Vel := 0;
   PRODUCT_TYPE[2].Motion.Gluing_Nozzle_X.Position[9].Pos := 0.0;
   PRODUCT_TYPE[2].Motion.Gluing_Nozzle_X.Position[9].Vel := 0;
   PRODUCT_TYPE[3].Motion.Gluing_Nozzle_X.Position[9].Pos := 0.0;
   PRODUCT_TYPE[3].Motion.Gluing_Nozzle_X.Position[9].Vel := 0;
   PRODUCT_TYPE[4].Motion.Gluing_Nozzle_X.Position[9].Pos := 0.0;
   PRODUCT_TYPE[4].Motion.Gluing_Nozzle_X.Position[9].Vel := 0;
   PRODUCT_TYPE[5].Motion.Gluing_Nozzle_X.Position[9].Pos := 0.0;
   PRODUCT_TYPE[5].Motion.Gluing_Nozzle_X.Position[9].Vel := 0;
   PRODUCT_TYPE[6].Motion.Gluing_Nozzle_X.Position[9].Pos := 0.0;
   PRODUCT_TYPE[6].Motion.Gluing_Nozzle_X.Position[9].Vel := 0;
   PRODUCT_TYPE[7].Motion.Gluing_Nozzle_X.Position[9].Pos := 0.0;
   PRODUCT_TYPE[7].Motion.Gluing_Nozzle_X.Position[9].Vel := 0;
   PRODUCT_TYPE[8].Motion.Gluing_Nozzle_X.Position[9].Pos := 0.0;
   PRODUCT_TYPE[8].Motion.Gluing_Nozzle_X.Position[9].Vel := 0;
   PRODUCT_TYPE[9].Motion.Gluing_Nozzle_X.Position[9].Pos := 0.0;
   PRODUCT_TYPE[9].Motion.Gluing_Nozzle_X.Position[9].Vel := 0;
   PRODUCT_TYPE[10].Motion.Gluing_Nozzle_X.Position[9].Pos := 0.0;
   PRODUCT_TYPE[10].Motion.Gluing_Nozzle_X.Position[9].Vel := 0;
   PRODUCT_TYPE[1].Motion.Gluing_Nozzle_X.Position[10].Pos := 0.0;
   PRODUCT_TYPE[1].Motion.Gluing_Nozzle_X.Position[10].Vel := 0;
   PRODUCT_TYPE[2].Motion.Gluing_Nozzle_X.Position[10].Pos := 0.0;
   PRODUCT_TYPE[2].Motion.Gluing_Nozzle_X.Position[10].Vel := 0;
   PRODUCT_TYPE[3].Motion.Gluing_Nozzle_X.Position[10].Pos := 0.0;
   PRODUCT_TYPE[3].Motion.Gluing_Nozzle_X.Position[10].Vel := 0;
   PRODUCT_TYPE[4].Motion.Gluing_Nozzle_X.Position[10].Pos := 0.0;
   PRODUCT_TYPE[4].Motion.Gluing_Nozzle_X.Position[10].Vel := 0;
   PRODUCT_TYPE[5].Motion.Gluing_Nozzle_X.Position[10].Pos := 0.0;
   PRODUCT_TYPE[5].Motion.Gluing_Nozzle_X.Position[10].Vel := 0;
   PRODUCT_TYPE[6].Motion.Gluing_Nozzle_X.Position[10].Pos := 0.0;
   PRODUCT_TYPE[6].Motion.Gluing_Nozzle_X.Position[10].Vel := 0;
   PRODUCT_TYPE[7].Motion.Gluing_Nozzle_X.Position[10].Pos := 0.0;
   PRODUCT_TYPE[7].Motion.Gluing_Nozzle_X.Position[10].Vel := 0;
   PRODUCT_TYPE[8].Motion.Gluing_Nozzle_X.Position[10].Pos := 0.0;
   PRODUCT_TYPE[8].Motion.Gluing_Nozzle_X.Position[10].Vel := 0;
   PRODUCT_TYPE[9].Motion.Gluing_Nozzle_X.Position[10].Pos := 0.0;
   PRODUCT_TYPE[9].Motion.Gluing_Nozzle_X.Position[10].Vel := 0;
   PRODUCT_TYPE[10].Motion.Gluing_Nozzle_X.Position[10].Pos := 0.0;
   PRODUCT_TYPE[10].Motion.Gluing_Nozzle_X.Position[10].Vel := 0;
   PRODUCT_TYPE[1].Motion.Gluing_Nozzle_X.Position[11].Pos := 0.0;
   PRODUCT_TYPE[1].Motion.Gluing_Nozzle_X.Position[11].Vel := 0;
   PRODUCT_TYPE[2].Motion.Gluing_Nozzle_X.Position[11].Pos := 0.0;
   PRODUCT_TYPE[2].Motion.Gluing_Nozzle_X.Position[11].Vel := 0;
   PRODUCT_TYPE[3].Motion.Gluing_Nozzle_X.Position[11].Pos := 0.0;
   PRODUCT_TYPE[3].Motion.Gluing_Nozzle_X.Position[11].Vel := 0;
   PRODUCT_TYPE[4].Motion.Gluing_Nozzle_X.Position[11].Pos := 0.0;
   PRODUCT_TYPE[4].Motion.Gluing_Nozzle_X.Position[11].Vel := 0;
   PRODUCT_TYPE[5].Motion.Gluing_Nozzle_X.Position[11].Pos := 0.0;
   PRODUCT_TYPE[5].Motion.Gluing_Nozzle_X.Position[11].Vel := 0;
   PRODUCT_TYPE[6].Motion.Gluing_Nozzle_X.Position[11].Pos := 0.0;
   PRODUCT_TYPE[6].Motion.Gluing_Nozzle_X.Position[11].Vel := 0;
   PRODUCT_TYPE[7].Motion.Gluing_Nozzle_X.Position[11].Pos := 0.0;
   PRODUCT_TYPE[7].Motion.Gluing_Nozzle_X.Position[11].Vel := 0;
   PRODUCT_TYPE[8].Motion.Gluing_Nozzle_X.Position[11].Pos := 0.0;
   PRODUCT_TYPE[8].Motion.Gluing_Nozzle_X.Position[11].Vel := 0;
   PRODUCT_TYPE[9].Motion.Gluing_Nozzle_X.Position[11].Pos := 0.0;
   PRODUCT_TYPE[9].Motion.Gluing_Nozzle_X.Position[11].Vel := 0;
   PRODUCT_TYPE[10].Motion.Gluing_Nozzle_X.Position[11].Pos := 0.0;
   PRODUCT_TYPE[10].Motion.Gluing_Nozzle_X.Position[11].Vel := 0;
   PRODUCT_TYPE[1].Motion.Gluing_Nozzle_X.Position[12].Pos := 0.0;
   PRODUCT_TYPE[1].Motion.Gluing_Nozzle_X.Position[12].Vel := 0;
   PRODUCT_TYPE[2].Motion.Gluing_Nozzle_X.Position[12].Pos := 0.0;
   PRODUCT_TYPE[2].Motion.Gluing_Nozzle_X.Position[12].Vel := 0;
   PRODUCT_TYPE[3].Motion.Gluing_Nozzle_X.Position[12].Pos := 0.0;
   PRODUCT_TYPE[3].Motion.Gluing_Nozzle_X.Position[12].Vel := 0;
   PRODUCT_TYPE[4].Motion.Gluing_Nozzle_X.Position[12].Pos := 0.0;
   PRODUCT_TYPE[4].Motion.Gluing_Nozzle_X.Position[12].Vel := 0;
   PRODUCT_TYPE[5].Motion.Gluing_Nozzle_X.Position[12].Pos := 0.0;
   PRODUCT_TYPE[5].Motion.Gluing_Nozzle_X.Position[12].Vel := 0;
   PRODUCT_TYPE[6].Motion.Gluing_Nozzle_X.Position[12].Pos := 0.0;
   PRODUCT_TYPE[6].Motion.Gluing_Nozzle_X.Position[12].Vel := 0;
   PRODUCT_TYPE[7].Motion.Gluing_Nozzle_X.Position[12].Pos := 0.0;
   PRODUCT_TYPE[7].Motion.Gluing_Nozzle_X.Position[12].Vel := 0;
   PRODUCT_TYPE[8].Motion.Gluing_Nozzle_X.Position[12].Pos := 0.0;
   PRODUCT_TYPE[8].Motion.Gluing_Nozzle_X.Position[12].Vel := 0;
   PRODUCT_TYPE[9].Motion.Gluing_Nozzle_X.Position[12].Pos := 0.0;
   PRODUCT_TYPE[9].Motion.Gluing_Nozzle_X.Position[12].Vel := 0;
   PRODUCT_TYPE[10].Motion.Gluing_Nozzle_X.Position[12].Pos := 0.0;
   PRODUCT_TYPE[10].Motion.Gluing_Nozzle_X.Position[12].Vel := 0;
   PRODUCT_TYPE[1].Motion.Gluing_Nozzle_X.Position[13].Pos := 0.0;
   PRODUCT_TYPE[1].Motion.Gluing_Nozzle_X.Position[13].Vel := 0;
   PRODUCT_TYPE[2].Motion.Gluing_Nozzle_X.Position[13].Pos := 0.0;
   PRODUCT_TYPE[2].Motion.Gluing_Nozzle_X.Position[13].Vel := 0;
   PRODUCT_TYPE[3].Motion.Gluing_Nozzle_X.Position[13].Pos := 0.0;
   PRODUCT_TYPE[3].Motion.Gluing_Nozzle_X.Position[13].Vel := 0;
   PRODUCT_TYPE[4].Motion.Gluing_Nozzle_X.Position[13].Pos := 0.0;
   PRODUCT_TYPE[4].Motion.Gluing_Nozzle_X.Position[13].Vel := 0;
   PRODUCT_TYPE[5].Motion.Gluing_Nozzle_X.Position[13].Pos := 0.0;
   PRODUCT_TYPE[5].Motion.Gluing_Nozzle_X.Position[13].Vel := 0;
   PRODUCT_TYPE[6].Motion.Gluing_Nozzle_X.Position[13].Pos := 0.0;
   PRODUCT_TYPE[6].Motion.Gluing_Nozzle_X.Position[13].Vel := 0;
   PRODUCT_TYPE[7].Motion.Gluing_Nozzle_X.Position[13].Pos := 0.0;
   PRODUCT_TYPE[7].Motion.Gluing_Nozzle_X.Position[13].Vel := 0;
   PRODUCT_TYPE[8].Motion.Gluing_Nozzle_X.Position[13].Pos := 0.0;
   PRODUCT_TYPE[8].Motion.Gluing_Nozzle_X.Position[13].Vel := 0;
   PRODUCT_TYPE[9].Motion.Gluing_Nozzle_X.Position[13].Pos := 0.0;
   PRODUCT_TYPE[9].Motion.Gluing_Nozzle_X.Position[13].Vel := 0;
   PRODUCT_TYPE[10].Motion.Gluing_Nozzle_X.Position[13].Pos := 0.0;
   PRODUCT_TYPE[10].Motion.Gluing_Nozzle_X.Position[13].Vel := 0;
   PRODUCT_TYPE[1].Motion.Gluing_Nozzle_X.Position[14].Pos := 0.0;
   PRODUCT_TYPE[1].Motion.Gluing_Nozzle_X.Position[14].Vel := 0;
   PRODUCT_TYPE[2].Motion.Gluing_Nozzle_X.Position[14].Pos := 0.0;
   PRODUCT_TYPE[2].Motion.Gluing_Nozzle_X.Position[14].Vel := 0;
   PRODUCT_TYPE[3].Motion.Gluing_Nozzle_X.Position[14].Pos := 0.0;
   PRODUCT_TYPE[3].Motion.Gluing_Nozzle_X.Position[14].Vel := 0;
   PRODUCT_TYPE[4].Motion.Gluing_Nozzle_X.Position[14].Pos := 0.0;
   PRODUCT_TYPE[4].Motion.Gluing_Nozzle_X.Position[14].Vel := 0;
   PRODUCT_TYPE[5].Motion.Gluing_Nozzle_X.Position[14].Pos := 0.0;
   PRODUCT_TYPE[5].Motion.Gluing_Nozzle_X.Position[14].Vel := 0;
   PRODUCT_TYPE[6].Motion.Gluing_Nozzle_X.Position[14].Pos := 0.0;
   PRODUCT_TYPE[6].Motion.Gluing_Nozzle_X.Position[14].Vel := 0;
   PRODUCT_TYPE[7].Motion.Gluing_Nozzle_X.Position[14].Pos := 0.0;
   PRODUCT_TYPE[7].Motion.Gluing_Nozzle_X.Position[14].Vel := 0;
   PRODUCT_TYPE[8].Motion.Gluing_Nozzle_X.Position[14].Pos := 0.0;
   PRODUCT_TYPE[8].Motion.Gluing_Nozzle_X.Position[14].Vel := 0;
   PRODUCT_TYPE[9].Motion.Gluing_Nozzle_X.Position[14].Pos := 0.0;
   PRODUCT_TYPE[9].Motion.Gluing_Nozzle_X.Position[14].Vel := 0;
   PRODUCT_TYPE[10].Motion.Gluing_Nozzle_X.Position[14].Pos := 0.0;
   PRODUCT_TYPE[10].Motion.Gluing_Nozzle_X.Position[14].Vel := 0;
   PRODUCT_TYPE[1].Motion.Gluing_Nozzle_X.Position[15].Pos := 0.0;
   PRODUCT_TYPE[1].Motion.Gluing_Nozzle_X.Position[15].Vel := 0;
   PRODUCT_TYPE[2].Motion.Gluing_Nozzle_X.Position[15].Pos := 0.0;
   PRODUCT_TYPE[2].Motion.Gluing_Nozzle_X.Position[15].Vel := 0;
   PRODUCT_TYPE[3].Motion.Gluing_Nozzle_X.Position[15].Pos := 0.0;
   PRODUCT_TYPE[3].Motion.Gluing_Nozzle_X.Position[15].Vel := 0;
   PRODUCT_TYPE[4].Motion.Gluing_Nozzle_X.Position[15].Pos := 0.0;
   PRODUCT_TYPE[4].Motion.Gluing_Nozzle_X.Position[15].Vel := 0;
   PRODUCT_TYPE[5].Motion.Gluing_Nozzle_X.Position[15].Pos := 0.0;
   PRODUCT_TYPE[5].Motion.Gluing_Nozzle_X.Position[15].Vel := 0;
   PRODUCT_TYPE[6].Motion.Gluing_Nozzle_X.Position[15].Pos := 0.0;
   PRODUCT_TYPE[6].Motion.Gluing_Nozzle_X.Position[15].Vel := 0;
   PRODUCT_TYPE[7].Motion.Gluing_Nozzle_X.Position[15].Pos := 0.0;
   PRODUCT_TYPE[7].Motion.Gluing_Nozzle_X.Position[15].Vel := 0;
   PRODUCT_TYPE[8].Motion.Gluing_Nozzle_X.Position[15].Pos := 0.0;
   PRODUCT_TYPE[8].Motion.Gluing_Nozzle_X.Position[15].Vel := 0;
   PRODUCT_TYPE[9].Motion.Gluing_Nozzle_X.Position[15].Pos := 0.0;
   PRODUCT_TYPE[9].Motion.Gluing_Nozzle_X.Position[15].Vel := 0;
   PRODUCT_TYPE[10].Motion.Gluing_Nozzle_X.Position[15].Pos := 0.0;
   PRODUCT_TYPE[10].Motion.Gluing_Nozzle_X.Position[15].Vel := 0;
   PRODUCT_TYPE[1].Motion.Gluing_Nozzle_X.Position[16].Pos := 0.0;
   PRODUCT_TYPE[1].Motion.Gluing_Nozzle_X.Position[16].Vel := 0;
   PRODUCT_TYPE[2].Motion.Gluing_Nozzle_X.Position[16].Pos := 0.0;
   PRODUCT_TYPE[2].Motion.Gluing_Nozzle_X.Position[16].Vel := 0;
   PRODUCT_TYPE[3].Motion.Gluing_Nozzle_X.Position[16].Pos := 0.0;
   PRODUCT_TYPE[3].Motion.Gluing_Nozzle_X.Position[16].Vel := 0;
   PRODUCT_TYPE[4].Motion.Gluing_Nozzle_X.Position[16].Pos := 0.0;
   PRODUCT_TYPE[4].Motion.Gluing_Nozzle_X.Position[16].Vel := 0;
   PRODUCT_TYPE[5].Motion.Gluing_Nozzle_X.Position[16].Pos := 0.0;
   PRODUCT_TYPE[5].Motion.Gluing_Nozzle_X.Position[16].Vel := 0;
   PRODUCT_TYPE[6].Motion.Gluing_Nozzle_X.Position[16].Pos := 0.0;
   PRODUCT_TYPE[6].Motion.Gluing_Nozzle_X.Position[16].Vel := 0;
   PRODUCT_TYPE[7].Motion.Gluing_Nozzle_X.Position[16].Pos := 0.0;
   PRODUCT_TYPE[7].Motion.Gluing_Nozzle_X.Position[16].Vel := 0;
   PRODUCT_TYPE[8].Motion.Gluing_Nozzle_X.Position[16].Pos := 0.0;
   PRODUCT_TYPE[8].Motion.Gluing_Nozzle_X.Position[16].Vel := 0;
   PRODUCT_TYPE[9].Motion.Gluing_Nozzle_X.Position[16].Pos := 0.0;
   PRODUCT_TYPE[9].Motion.Gluing_Nozzle_X.Position[16].Vel := 0;
   PRODUCT_TYPE[10].Motion.Gluing_Nozzle_X.Position[16].Pos := 0.0;
   PRODUCT_TYPE[10].Motion.Gluing_Nozzle_X.Position[16].Vel := 0;
   PRODUCT_TYPE[1].Motion.Gluing_Nozzle_X.Position[17].Pos := 0.0;
   PRODUCT_TYPE[1].Motion.Gluing_Nozzle_X.Position[17].Vel := 0;
   PRODUCT_TYPE[2].Motion.Gluing_Nozzle_X.Position[17].Pos := 0.0;
   PRODUCT_TYPE[2].Motion.Gluing_Nozzle_X.Position[17].Vel := 0;
   PRODUCT_TYPE[3].Motion.Gluing_Nozzle_X.Position[17].Pos := 0.0;
   PRODUCT_TYPE[3].Motion.Gluing_Nozzle_X.Position[17].Vel := 0;
   PRODUCT_TYPE[4].Motion.Gluing_Nozzle_X.Position[17].Pos := 0.0;
   PRODUCT_TYPE[4].Motion.Gluing_Nozzle_X.Position[17].Vel := 0;
   PRODUCT_TYPE[5].Motion.Gluing_Nozzle_X.Position[17].Pos := 0.0;
   PRODUCT_TYPE[5].Motion.Gluing_Nozzle_X.Position[17].Vel := 0;
   PRODUCT_TYPE[6].Motion.Gluing_Nozzle_X.Position[17].Pos := 0.0;
   PRODUCT_TYPE[6].Motion.Gluing_Nozzle_X.Position[17].Vel := 0;
   PRODUCT_TYPE[7].Motion.Gluing_Nozzle_X.Position[17].Pos := 0.0;
   PRODUCT_TYPE[7].Motion.Gluing_Nozzle_X.Position[17].Vel := 0;
   PRODUCT_TYPE[8].Motion.Gluing_Nozzle_X.Position[17].Pos := 0.0;
   PRODUCT_TYPE[8].Motion.Gluing_Nozzle_X.Position[17].Vel := 0;
   PRODUCT_TYPE[9].Motion.Gluing_Nozzle_X.Position[17].Pos := 0.0;
   PRODUCT_TYPE[9].Motion.Gluing_Nozzle_X.Position[17].Vel := 0;
   PRODUCT_TYPE[10].Motion.Gluing_Nozzle_X.Position[17].Pos := 0.0;
   PRODUCT_TYPE[10].Motion.Gluing_Nozzle_X.Position[17].Vel := 0;
   PRODUCT_TYPE[1].Motion.Gluing_Nozzle_X.Position[18].Pos := 0.0;
   PRODUCT_TYPE[1].Motion.Gluing_Nozzle_X.Position[18].Vel := 0;
   PRODUCT_TYPE[2].Motion.Gluing_Nozzle_X.Position[18].Pos := 0.0;
   PRODUCT_TYPE[2].Motion.Gluing_Nozzle_X.Position[18].Vel := 0;
   PRODUCT_TYPE[3].Motion.Gluing_Nozzle_X.Position[18].Pos := 0.0;
   PRODUCT_TYPE[3].Motion.Gluing_Nozzle_X.Position[18].Vel := 0;
   PRODUCT_TYPE[4].Motion.Gluing_Nozzle_X.Position[18].Pos := 0.0;
   PRODUCT_TYPE[4].Motion.Gluing_Nozzle_X.Position[18].Vel := 0;
   PRODUCT_TYPE[5].Motion.Gluing_Nozzle_X.Position[18].Pos := 0.0;
   PRODUCT_TYPE[5].Motion.Gluing_Nozzle_X.Position[18].Vel := 0;
   PRODUCT_TYPE[6].Motion.Gluing_Nozzle_X.Position[18].Pos := 0.0;
   PRODUCT_TYPE[6].Motion.Gluing_Nozzle_X.Position[18].Vel := 0;
   PRODUCT_TYPE[7].Motion.Gluing_Nozzle_X.Position[18].Pos := 0.0;
   PRODUCT_TYPE[7].Motion.Gluing_Nozzle_X.Position[18].Vel := 0;
   PRODUCT_TYPE[8].Motion.Gluing_Nozzle_X.Position[18].Pos := 0.0;
   PRODUCT_TYPE[8].Motion.Gluing_Nozzle_X.Position[18].Vel := 0;
   PRODUCT_TYPE[9].Motion.Gluing_Nozzle_X.Position[18].Pos := 0.0;
   PRODUCT_TYPE[9].Motion.Gluing_Nozzle_X.Position[18].Vel := 0;
   PRODUCT_TYPE[10].Motion.Gluing_Nozzle_X.Position[18].Pos := 0.0;
   PRODUCT_TYPE[10].Motion.Gluing_Nozzle_X.Position[18].Vel := 0;
   PRODUCT_TYPE[1].Motion.Gluing_Nozzle_X.Position[19].Pos := 0.0;
   PRODUCT_TYPE[1].Motion.Gluing_Nozzle_X.Position[19].Vel := 0;
   PRODUCT_TYPE[2].Motion.Gluing_Nozzle_X.Position[19].Pos := 0.0;
   PRODUCT_TYPE[2].Motion.Gluing_Nozzle_X.Position[19].Vel := 0;
   PRODUCT_TYPE[3].Motion.Gluing_Nozzle_X.Position[19].Pos := 0.0;
   PRODUCT_TYPE[3].Motion.Gluing_Nozzle_X.Position[19].Vel := 0;
   PRODUCT_TYPE[4].Motion.Gluing_Nozzle_X.Position[19].Pos := 0.0;
   PRODUCT_TYPE[4].Motion.Gluing_Nozzle_X.Position[19].Vel := 0;
   PRODUCT_TYPE[5].Motion.Gluing_Nozzle_X.Position[19].Pos := 0.0;
   PRODUCT_TYPE[5].Motion.Gluing_Nozzle_X.Position[19].Vel := 0;
   PRODUCT_TYPE[6].Motion.Gluing_Nozzle_X.Position[19].Pos := 0.0;
   PRODUCT_TYPE[6].Motion.Gluing_Nozzle_X.Position[19].Vel := 0;
   PRODUCT_TYPE[7].Motion.Gluing_Nozzle_X.Position[19].Pos := 0.0;
   PRODUCT_TYPE[7].Motion.Gluing_Nozzle_X.Position[19].Vel := 0;
   PRODUCT_TYPE[8].Motion.Gluing_Nozzle_X.Position[19].Pos := 0.0;
   PRODUCT_TYPE[8].Motion.Gluing_Nozzle_X.Position[19].Vel := 0;
   PRODUCT_TYPE[9].Motion.Gluing_Nozzle_X.Position[19].Pos := 0.0;
   PRODUCT_TYPE[9].Motion.Gluing_Nozzle_X.Position[19].Vel := 0;
   PRODUCT_TYPE[10].Motion.Gluing_Nozzle_X.Position[19].Pos := 0.0;
   PRODUCT_TYPE[10].Motion.Gluing_Nozzle_X.Position[19].Vel := 0;
   PRODUCT_TYPE[1].Motion.Gluing_Nozzle_X.Position[20].Pos := 0.0;
   PRODUCT_TYPE[1].Motion.Gluing_Nozzle_X.Position[20].Vel := 0;
   PRODUCT_TYPE[2].Motion.Gluing_Nozzle_X.Position[20].Pos := 0.0;
   PRODUCT_TYPE[2].Motion.Gluing_Nozzle_X.Position[20].Vel := 0;
   PRODUCT_TYPE[3].Motion.Gluing_Nozzle_X.Position[20].Pos := 0.0;
   PRODUCT_TYPE[3].Motion.Gluing_Nozzle_X.Position[20].Vel := 0;
   PRODUCT_TYPE[4].Motion.Gluing_Nozzle_X.Position[20].Pos := 0.0;
   PRODUCT_TYPE[4].Motion.Gluing_Nozzle_X.Position[20].Vel := 0;
   PRODUCT_TYPE[5].Motion.Gluing_Nozzle_X.Position[20].Pos := 0.0;
   PRODUCT_TYPE[5].Motion.Gluing_Nozzle_X.Position[20].Vel := 0;
   PRODUCT_TYPE[6].Motion.Gluing_Nozzle_X.Position[20].Pos := 0.0;
   PRODUCT_TYPE[6].Motion.Gluing_Nozzle_X.Position[20].Vel := 0;
   PRODUCT_TYPE[7].Motion.Gluing_Nozzle_X.Position[20].Pos := 0.0;
   PRODUCT_TYPE[7].Motion.Gluing_Nozzle_X.Position[20].Vel := 0;
   PRODUCT_TYPE[8].Motion.Gluing_Nozzle_X.Position[20].Pos := 0.0;
   PRODUCT_TYPE[8].Motion.Gluing_Nozzle_X.Position[20].Vel := 0;
   PRODUCT_TYPE[9].Motion.Gluing_Nozzle_X.Position[20].Pos := 0.0;
   PRODUCT_TYPE[9].Motion.Gluing_Nozzle_X.Position[20].Vel := 0;
   PRODUCT_TYPE[10].Motion.Gluing_Nozzle_X.Position[20].Pos := 0.0;
   PRODUCT_TYPE[10].Motion.Gluing_Nozzle_X.Position[20].Vel := 0;
   PRODUCT_TYPE[1].Motion.Gluing_Nozzle_Y.Position[1].Pos := 115.47;
   PRODUCT_TYPE[1].Motion.Gluing_Nozzle_Y.Position[1].Vel := 200;
   PRODUCT_TYPE[2].Motion.Gluing_Nozzle_Y.Position[1].Pos := 115.47;
   PRODUCT_TYPE[2].Motion.Gluing_Nozzle_Y.Position[1].Vel := 200;
   PRODUCT_TYPE[3].Motion.Gluing_Nozzle_Y.Position[1].Pos := 115.47;
   PRODUCT_TYPE[3].Motion.Gluing_Nozzle_Y.Position[1].Vel := 200;
   PRODUCT_TYPE[4].Motion.Gluing_Nozzle_Y.Position[1].Pos := 115.47;
   PRODUCT_TYPE[4].Motion.Gluing_Nozzle_Y.Position[1].Vel := 200;
   PRODUCT_TYPE[5].Motion.Gluing_Nozzle_Y.Position[1].Pos := 115.47;
   PRODUCT_TYPE[5].Motion.Gluing_Nozzle_Y.Position[1].Vel := 200;
   PRODUCT_TYPE[6].Motion.Gluing_Nozzle_Y.Position[1].Pos := 115.47;
   PRODUCT_TYPE[6].Motion.Gluing_Nozzle_Y.Position[1].Vel := 200;
   PRODUCT_TYPE[7].Motion.Gluing_Nozzle_Y.Position[1].Pos := 115.47;
   PRODUCT_TYPE[7].Motion.Gluing_Nozzle_Y.Position[1].Vel := 200;
   PRODUCT_TYPE[8].Motion.Gluing_Nozzle_Y.Position[1].Pos := 115.47;
   PRODUCT_TYPE[8].Motion.Gluing_Nozzle_Y.Position[1].Vel := 200;
   PRODUCT_TYPE[9].Motion.Gluing_Nozzle_Y.Position[1].Pos := 115.47;
   PRODUCT_TYPE[9].Motion.Gluing_Nozzle_Y.Position[1].Vel := 200;
   PRODUCT_TYPE[10].Motion.Gluing_Nozzle_Y.Position[1].Pos := 115.47;
   PRODUCT_TYPE[10].Motion.Gluing_Nozzle_Y.Position[1].Vel := 200;
   PRODUCT_TYPE[1].Motion.Gluing_Nozzle_Y.Position[2].Pos := 115.47;
   PRODUCT_TYPE[1].Motion.Gluing_Nozzle_Y.Position[2].Vel := 200;
   PRODUCT_TYPE[2].Motion.Gluing_Nozzle_Y.Position[2].Pos := 115.47;
   PRODUCT_TYPE[2].Motion.Gluing_Nozzle_Y.Position[2].Vel := 200;
   PRODUCT_TYPE[3].Motion.Gluing_Nozzle_Y.Position[2].Pos := 115.47;
   PRODUCT_TYPE[3].Motion.Gluing_Nozzle_Y.Position[2].Vel := 200;
   PRODUCT_TYPE[4].Motion.Gluing_Nozzle_Y.Position[2].Pos := 115.47;
   PRODUCT_TYPE[4].Motion.Gluing_Nozzle_Y.Position[2].Vel := 200;
   PRODUCT_TYPE[5].Motion.Gluing_Nozzle_Y.Position[2].Pos := 115.47;
   PRODUCT_TYPE[5].Motion.Gluing_Nozzle_Y.Position[2].Vel := 200;
   PRODUCT_TYPE[6].Motion.Gluing_Nozzle_Y.Position[2].Pos := 115.47;
   PRODUCT_TYPE[6].Motion.Gluing_Nozzle_Y.Position[2].Vel := 200;
   PRODUCT_TYPE[7].Motion.Gluing_Nozzle_Y.Position[2].Pos := 115.47;
   PRODUCT_TYPE[7].Motion.Gluing_Nozzle_Y.Position[2].Vel := 200;
   PRODUCT_TYPE[8].Motion.Gluing_Nozzle_Y.Position[2].Pos := 115.47;
   PRODUCT_TYPE[8].Motion.Gluing_Nozzle_Y.Position[2].Vel := 200;
   PRODUCT_TYPE[9].Motion.Gluing_Nozzle_Y.Position[2].Pos := 115.47;
   PRODUCT_TYPE[9].Motion.Gluing_Nozzle_Y.Position[2].Vel := 200;
   PRODUCT_TYPE[10].Motion.Gluing_Nozzle_Y.Position[2].Pos := 115.47;
   PRODUCT_TYPE[10].Motion.Gluing_Nozzle_Y.Position[2].Vel := 200;
   PRODUCT_TYPE[1].Motion.Gluing_Nozzle_Y.Position[3].Pos := 115.47;
   PRODUCT_TYPE[1].Motion.Gluing_Nozzle_Y.Position[3].Vel := 200;
   PRODUCT_TYPE[2].Motion.Gluing_Nozzle_Y.Position[3].Pos := 115.47;
   PRODUCT_TYPE[2].Motion.Gluing_Nozzle_Y.Position[3].Vel := 200;
   PRODUCT_TYPE[3].Motion.Gluing_Nozzle_Y.Position[3].Pos := 115.47;
   PRODUCT_TYPE[3].Motion.Gluing_Nozzle_Y.Position[3].Vel := 200;
   PRODUCT_TYPE[4].Motion.Gluing_Nozzle_Y.Position[3].Pos := 115.47;
   PRODUCT_TYPE[4].Motion.Gluing_Nozzle_Y.Position[3].Vel := 200;
   PRODUCT_TYPE[5].Motion.Gluing_Nozzle_Y.Position[3].Pos := 115.47;
   PRODUCT_TYPE[5].Motion.Gluing_Nozzle_Y.Position[3].Vel := 200;
   PRODUCT_TYPE[6].Motion.Gluing_Nozzle_Y.Position[3].Pos := 115.47;
   PRODUCT_TYPE[6].Motion.Gluing_Nozzle_Y.Position[3].Vel := 200;
   PRODUCT_TYPE[7].Motion.Gluing_Nozzle_Y.Position[3].Pos := 115.47;
   PRODUCT_TYPE[7].Motion.Gluing_Nozzle_Y.Position[3].Vel := 200;
   PRODUCT_TYPE[8].Motion.Gluing_Nozzle_Y.Position[3].Pos := 115.47;
   PRODUCT_TYPE[8].Motion.Gluing_Nozzle_Y.Position[3].Vel := 200;
   PRODUCT_TYPE[9].Motion.Gluing_Nozzle_Y.Position[3].Pos := 115.47;
   PRODUCT_TYPE[9].Motion.Gluing_Nozzle_Y.Position[3].Vel := 200;
   PRODUCT_TYPE[10].Motion.Gluing_Nozzle_Y.Position[3].Pos := 115.47;
   PRODUCT_TYPE[10].Motion.Gluing_Nozzle_Y.Position[3].Vel := 200;
   PRODUCT_TYPE[1].Motion.Gluing_Nozzle_Y.Position[4].Pos := 115.47;
   PRODUCT_TYPE[1].Motion.Gluing_Nozzle_Y.Position[4].Vel := 200;
   PRODUCT_TYPE[2].Motion.Gluing_Nozzle_Y.Position[4].Pos := 115.47;
   PRODUCT_TYPE[2].Motion.Gluing_Nozzle_Y.Position[4].Vel := 200;
   PRODUCT_TYPE[3].Motion.Gluing_Nozzle_Y.Position[4].Pos := 115.47;
   PRODUCT_TYPE[3].Motion.Gluing_Nozzle_Y.Position[4].Vel := 200;
   PRODUCT_TYPE[4].Motion.Gluing_Nozzle_Y.Position[4].Pos := 115.47;
   PRODUCT_TYPE[4].Motion.Gluing_Nozzle_Y.Position[4].Vel := 200;
   PRODUCT_TYPE[5].Motion.Gluing_Nozzle_Y.Position[4].Pos := 115.47;
   PRODUCT_TYPE[5].Motion.Gluing_Nozzle_Y.Position[4].Vel := 200;
   PRODUCT_TYPE[6].Motion.Gluing_Nozzle_Y.Position[4].Pos := 115.47;
   PRODUCT_TYPE[6].Motion.Gluing_Nozzle_Y.Position[4].Vel := 200;
   PRODUCT_TYPE[7].Motion.Gluing_Nozzle_Y.Position[4].Pos := 115.47;
   PRODUCT_TYPE[7].Motion.Gluing_Nozzle_Y.Position[4].Vel := 200;
   PRODUCT_TYPE[8].Motion.Gluing_Nozzle_Y.Position[4].Pos := 115.47;
   PRODUCT_TYPE[8].Motion.Gluing_Nozzle_Y.Position[4].Vel := 200;
   PRODUCT_TYPE[9].Motion.Gluing_Nozzle_Y.Position[4].Pos := 115.47;
   PRODUCT_TYPE[9].Motion.Gluing_Nozzle_Y.Position[4].Vel := 200;
   PRODUCT_TYPE[10].Motion.Gluing_Nozzle_Y.Position[4].Pos := 115.47;
   PRODUCT_TYPE[10].Motion.Gluing_Nozzle_Y.Position[4].Vel := 200;
   PRODUCT_TYPE[1].Motion.Gluing_Nozzle_Y.Position[5].Pos := 115.47;
   PRODUCT_TYPE[1].Motion.Gluing_Nozzle_Y.Position[5].Vel := 200;
   PRODUCT_TYPE[2].Motion.Gluing_Nozzle_Y.Position[5].Pos := 115.47;
   PRODUCT_TYPE[2].Motion.Gluing_Nozzle_Y.Position[5].Vel := 200;
   PRODUCT_TYPE[3].Motion.Gluing_Nozzle_Y.Position[5].Pos := 115.47;
   PRODUCT_TYPE[3].Motion.Gluing_Nozzle_Y.Position[5].Vel := 200;
   PRODUCT_TYPE[4].Motion.Gluing_Nozzle_Y.Position[5].Pos := 115.47;
   PRODUCT_TYPE[4].Motion.Gluing_Nozzle_Y.Position[5].Vel := 200;
   PRODUCT_TYPE[5].Motion.Gluing_Nozzle_Y.Position[5].Pos := 115.47;
   PRODUCT_TYPE[5].Motion.Gluing_Nozzle_Y.Position[5].Vel := 200;
   PRODUCT_TYPE[6].Motion.Gluing_Nozzle_Y.Position[5].Pos := 115.47;
   PRODUCT_TYPE[6].Motion.Gluing_Nozzle_Y.Position[5].Vel := 200;
   PRODUCT_TYPE[7].Motion.Gluing_Nozzle_Y.Position[5].Pos := 115.47;
   PRODUCT_TYPE[7].Motion.Gluing_Nozzle_Y.Position[5].Vel := 200;
   PRODUCT_TYPE[8].Motion.Gluing_Nozzle_Y.Position[5].Pos := 115.47;
   PRODUCT_TYPE[8].Motion.Gluing_Nozzle_Y.Position[5].Vel := 200;
   PRODUCT_TYPE[9].Motion.Gluing_Nozzle_Y.Position[5].Pos := 115.47;
   PRODUCT_TYPE[9].Motion.Gluing_Nozzle_Y.Position[5].Vel := 200;
   PRODUCT_TYPE[10].Motion.Gluing_Nozzle_Y.Position[5].Pos := 115.47;
   PRODUCT_TYPE[10].Motion.Gluing_Nozzle_Y.Position[5].Vel := 200;
   PRODUCT_TYPE[1].Motion.Gluing_Nozzle_Y.Position[6].Pos := 110.18;
   PRODUCT_TYPE[1].Motion.Gluing_Nozzle_Y.Position[6].Vel := 200;
   PRODUCT_TYPE[2].Motion.Gluing_Nozzle_Y.Position[6].Pos := 110.18;
   PRODUCT_TYPE[2].Motion.Gluing_Nozzle_Y.Position[6].Vel := 200;
   PRODUCT_TYPE[3].Motion.Gluing_Nozzle_Y.Position[6].Pos := 110.18;
   PRODUCT_TYPE[3].Motion.Gluing_Nozzle_Y.Position[6].Vel := 200;
   PRODUCT_TYPE[4].Motion.Gluing_Nozzle_Y.Position[6].Pos := 110.18;
   PRODUCT_TYPE[4].Motion.Gluing_Nozzle_Y.Position[6].Vel := 200;
   PRODUCT_TYPE[5].Motion.Gluing_Nozzle_Y.Position[6].Pos := 110.18;
   PRODUCT_TYPE[5].Motion.Gluing_Nozzle_Y.Position[6].Vel := 200;
   PRODUCT_TYPE[6].Motion.Gluing_Nozzle_Y.Position[6].Pos := 110.18;
   PRODUCT_TYPE[6].Motion.Gluing_Nozzle_Y.Position[6].Vel := 200;
   PRODUCT_TYPE[7].Motion.Gluing_Nozzle_Y.Position[6].Pos := 110.18;
   PRODUCT_TYPE[7].Motion.Gluing_Nozzle_Y.Position[6].Vel := 200;
   PRODUCT_TYPE[8].Motion.Gluing_Nozzle_Y.Position[6].Pos := 110.18;
   PRODUCT_TYPE[8].Motion.Gluing_Nozzle_Y.Position[6].Vel := 200;
   PRODUCT_TYPE[9].Motion.Gluing_Nozzle_Y.Position[6].Pos := 110.18;
   PRODUCT_TYPE[9].Motion.Gluing_Nozzle_Y.Position[6].Vel := 200;
   PRODUCT_TYPE[10].Motion.Gluing_Nozzle_Y.Position[6].Pos := 110.18;
   PRODUCT_TYPE[10].Motion.Gluing_Nozzle_Y.Position[6].Vel := 200;
   PRODUCT_TYPE[1].Motion.Gluing_Nozzle_Y.Position[7].Pos := 60.52;
   PRODUCT_TYPE[1].Motion.Gluing_Nozzle_Y.Position[7].Vel := 200;
   PRODUCT_TYPE[2].Motion.Gluing_Nozzle_Y.Position[7].Pos := 60.52;
   PRODUCT_TYPE[2].Motion.Gluing_Nozzle_Y.Position[7].Vel := 200;
   PRODUCT_TYPE[3].Motion.Gluing_Nozzle_Y.Position[7].Pos := 60.52;
   PRODUCT_TYPE[3].Motion.Gluing_Nozzle_Y.Position[7].Vel := 200;
   PRODUCT_TYPE[4].Motion.Gluing_Nozzle_Y.Position[7].Pos := 60.52;
   PRODUCT_TYPE[4].Motion.Gluing_Nozzle_Y.Position[7].Vel := 200;
   PRODUCT_TYPE[5].Motion.Gluing_Nozzle_Y.Position[7].Pos := 60.52;
   PRODUCT_TYPE[5].Motion.Gluing_Nozzle_Y.Position[7].Vel := 200;
   PRODUCT_TYPE[6].Motion.Gluing_Nozzle_Y.Position[7].Pos := 60.52;
   PRODUCT_TYPE[6].Motion.Gluing_Nozzle_Y.Position[7].Vel := 200;
   PRODUCT_TYPE[7].Motion.Gluing_Nozzle_Y.Position[7].Pos := 60.52;
   PRODUCT_TYPE[7].Motion.Gluing_Nozzle_Y.Position[7].Vel := 200;
   PRODUCT_TYPE[8].Motion.Gluing_Nozzle_Y.Position[7].Pos := 60.52;
   PRODUCT_TYPE[8].Motion.Gluing_Nozzle_Y.Position[7].Vel := 200;
   PRODUCT_TYPE[9].Motion.Gluing_Nozzle_Y.Position[7].Pos := 60.52;
   PRODUCT_TYPE[9].Motion.Gluing_Nozzle_Y.Position[7].Vel := 200;
   PRODUCT_TYPE[10].Motion.Gluing_Nozzle_Y.Position[7].Pos := 60.52;
   PRODUCT_TYPE[10].Motion.Gluing_Nozzle_Y.Position[7].Vel := 200;
   PRODUCT_TYPE[1].Motion.Gluing_Nozzle_Y.Position[8].Pos := 80.0;
   PRODUCT_TYPE[1].Motion.Gluing_Nozzle_Y.Position[8].Vel := 100;
   PRODUCT_TYPE[2].Motion.Gluing_Nozzle_Y.Position[8].Pos := 80.0;
   PRODUCT_TYPE[2].Motion.Gluing_Nozzle_Y.Position[8].Vel := 100;
   PRODUCT_TYPE[3].Motion.Gluing_Nozzle_Y.Position[8].Pos := 80.0;
   PRODUCT_TYPE[3].Motion.Gluing_Nozzle_Y.Position[8].Vel := 100;
   PRODUCT_TYPE[4].Motion.Gluing_Nozzle_Y.Position[8].Pos := 80.0;
   PRODUCT_TYPE[4].Motion.Gluing_Nozzle_Y.Position[8].Vel := 100;
   PRODUCT_TYPE[5].Motion.Gluing_Nozzle_Y.Position[8].Pos := 80.0;
   PRODUCT_TYPE[5].Motion.Gluing_Nozzle_Y.Position[8].Vel := 100;
   PRODUCT_TYPE[6].Motion.Gluing_Nozzle_Y.Position[8].Pos := 80.0;
   PRODUCT_TYPE[6].Motion.Gluing_Nozzle_Y.Position[8].Vel := 100;
   PRODUCT_TYPE[7].Motion.Gluing_Nozzle_Y.Position[8].Pos := 80.0;
   PRODUCT_TYPE[7].Motion.Gluing_Nozzle_Y.Position[8].Vel := 100;
   PRODUCT_TYPE[8].Motion.Gluing_Nozzle_Y.Position[8].Pos := 80.0;
   PRODUCT_TYPE[8].Motion.Gluing_Nozzle_Y.Position[8].Vel := 100;
   PRODUCT_TYPE[9].Motion.Gluing_Nozzle_Y.Position[8].Pos := 80.0;
   PRODUCT_TYPE[9].Motion.Gluing_Nozzle_Y.Position[8].Vel := 100;
   PRODUCT_TYPE[10].Motion.Gluing_Nozzle_Y.Position[8].Pos := 80.0;
   PRODUCT_TYPE[10].Motion.Gluing_Nozzle_Y.Position[8].Vel := 100;
   PRODUCT_TYPE[1].Motion.Gluing_Nozzle_Y.Position[9].Pos := 0.0;
   PRODUCT_TYPE[1].Motion.Gluing_Nozzle_Y.Position[9].Vel := 0;
   PRODUCT_TYPE[2].Motion.Gluing_Nozzle_Y.Position[9].Pos := 0.0;
   PRODUCT_TYPE[2].Motion.Gluing_Nozzle_Y.Position[9].Vel := 0;
   PRODUCT_TYPE[3].Motion.Gluing_Nozzle_Y.Position[9].Pos := 0.0;
   PRODUCT_TYPE[3].Motion.Gluing_Nozzle_Y.Position[9].Vel := 0;
   PRODUCT_TYPE[4].Motion.Gluing_Nozzle_Y.Position[9].Pos := 0.0;
   PRODUCT_TYPE[4].Motion.Gluing_Nozzle_Y.Position[9].Vel := 0;
   PRODUCT_TYPE[5].Motion.Gluing_Nozzle_Y.Position[9].Pos := 0.0;
   PRODUCT_TYPE[5].Motion.Gluing_Nozzle_Y.Position[9].Vel := 0;
   PRODUCT_TYPE[6].Motion.Gluing_Nozzle_Y.Position[9].Pos := 0.0;
   PRODUCT_TYPE[6].Motion.Gluing_Nozzle_Y.Position[9].Vel := 0;
   PRODUCT_TYPE[7].Motion.Gluing_Nozzle_Y.Position[9].Pos := 0.0;
   PRODUCT_TYPE[7].Motion.Gluing_Nozzle_Y.Position[9].Vel := 0;
   PRODUCT_TYPE[8].Motion.Gluing_Nozzle_Y.Position[9].Pos := 0.0;
   PRODUCT_TYPE[8].Motion.Gluing_Nozzle_Y.Position[9].Vel := 0;
   PRODUCT_TYPE[9].Motion.Gluing_Nozzle_Y.Position[9].Pos := 0.0;
   PRODUCT_TYPE[9].Motion.Gluing_Nozzle_Y.Position[9].Vel := 0;
   PRODUCT_TYPE[10].Motion.Gluing_Nozzle_Y.Position[9].Pos := 0.0;
   PRODUCT_TYPE[10].Motion.Gluing_Nozzle_Y.Position[9].Vel := 0;
   PRODUCT_TYPE[1].Motion.Gluing_Nozzle_Y.Position[10].Pos := 0.0;
   PRODUCT_TYPE[1].Motion.Gluing_Nozzle_Y.Position[10].Vel := 0;
   PRODUCT_TYPE[2].Motion.Gluing_Nozzle_Y.Position[10].Pos := 0.0;
   PRODUCT_TYPE[2].Motion.Gluing_Nozzle_Y.Position[10].Vel := 0;
   PRODUCT_TYPE[3].Motion.Gluing_Nozzle_Y.Position[10].Pos := 0.0;
   PRODUCT_TYPE[3].Motion.Gluing_Nozzle_Y.Position[10].Vel := 0;
   PRODUCT_TYPE[4].Motion.Gluing_Nozzle_Y.Position[10].Pos := 0.0;
   PRODUCT_TYPE[4].Motion.Gluing_Nozzle_Y.Position[10].Vel := 0;
   PRODUCT_TYPE[5].Motion.Gluing_Nozzle_Y.Position[10].Pos := 0.0;
   PRODUCT_TYPE[5].Motion.Gluing_Nozzle_Y.Position[10].Vel := 0;
   PRODUCT_TYPE[6].Motion.Gluing_Nozzle_Y.Position[10].Pos := 0.0;
   PRODUCT_TYPE[6].Motion.Gluing_Nozzle_Y.Position[10].Vel := 0;
   PRODUCT_TYPE[7].Motion.Gluing_Nozzle_Y.Position[10].Pos := 0.0;
   PRODUCT_TYPE[7].Motion.Gluing_Nozzle_Y.Position[10].Vel := 0;
   PRODUCT_TYPE[8].Motion.Gluing_Nozzle_Y.Position[10].Pos := 0.0;
   PRODUCT_TYPE[8].Motion.Gluing_Nozzle_Y.Position[10].Vel := 0;
   PRODUCT_TYPE[9].Motion.Gluing_Nozzle_Y.Position[10].Pos := 0.0;
   PRODUCT_TYPE[9].Motion.Gluing_Nozzle_Y.Position[10].Vel := 0;
   PRODUCT_TYPE[10].Motion.Gluing_Nozzle_Y.Position[10].Pos := 0.0;
   PRODUCT_TYPE[10].Motion.Gluing_Nozzle_Y.Position[10].Vel := 0;
   PRODUCT_TYPE[1].Motion.Gluing_Nozzle_Y.Position[11].Pos := 0.0;
   PRODUCT_TYPE[1].Motion.Gluing_Nozzle_Y.Position[11].Vel := 0;
   PRODUCT_TYPE[2].Motion.Gluing_Nozzle_Y.Position[11].Pos := 0.0;
   PRODUCT_TYPE[2].Motion.Gluing_Nozzle_Y.Position[11].Vel := 0;
   PRODUCT_TYPE[3].Motion.Gluing_Nozzle_Y.Position[11].Pos := 0.0;
   PRODUCT_TYPE[3].Motion.Gluing_Nozzle_Y.Position[11].Vel := 0;
   PRODUCT_TYPE[4].Motion.Gluing_Nozzle_Y.Position[11].Pos := 0.0;
   PRODUCT_TYPE[4].Motion.Gluing_Nozzle_Y.Position[11].Vel := 0;
   PRODUCT_TYPE[5].Motion.Gluing_Nozzle_Y.Position[11].Pos := 0.0;
   PRODUCT_TYPE[5].Motion.Gluing_Nozzle_Y.Position[11].Vel := 0;
   PRODUCT_TYPE[6].Motion.Gluing_Nozzle_Y.Position[11].Pos := 0.0;
   PRODUCT_TYPE[6].Motion.Gluing_Nozzle_Y.Position[11].Vel := 0;
   PRODUCT_TYPE[7].Motion.Gluing_Nozzle_Y.Position[11].Pos := 0.0;
   PRODUCT_TYPE[7].Motion.Gluing_Nozzle_Y.Position[11].Vel := 0;
   PRODUCT_TYPE[8].Motion.Gluing_Nozzle_Y.Position[11].Pos := 0.0;
   PRODUCT_TYPE[8].Motion.Gluing_Nozzle_Y.Position[11].Vel := 0;
   PRODUCT_TYPE[9].Motion.Gluing_Nozzle_Y.Position[11].Pos := 0.0;
   PRODUCT_TYPE[9].Motion.Gluing_Nozzle_Y.Position[11].Vel := 0;
   PRODUCT_TYPE[10].Motion.Gluing_Nozzle_Y.Position[11].Pos := 0.0;
   PRODUCT_TYPE[10].Motion.Gluing_Nozzle_Y.Position[11].Vel := 0;
   PRODUCT_TYPE[1].Motion.Gluing_Nozzle_Y.Position[12].Pos := 0.0;
   PRODUCT_TYPE[1].Motion.Gluing_Nozzle_Y.Position[12].Vel := 0;
   PRODUCT_TYPE[2].Motion.Gluing_Nozzle_Y.Position[12].Pos := 0.0;
   PRODUCT_TYPE[2].Motion.Gluing_Nozzle_Y.Position[12].Vel := 0;
   PRODUCT_TYPE[3].Motion.Gluing_Nozzle_Y.Position[12].Pos := 0.0;
   PRODUCT_TYPE[3].Motion.Gluing_Nozzle_Y.Position[12].Vel := 0;
   PRODUCT_TYPE[4].Motion.Gluing_Nozzle_Y.Position[12].Pos := 0.0;
   PRODUCT_TYPE[4].Motion.Gluing_Nozzle_Y.Position[12].Vel := 0;
   PRODUCT_TYPE[5].Motion.Gluing_Nozzle_Y.Position[12].Pos := 0.0;
   PRODUCT_TYPE[5].Motion.Gluing_Nozzle_Y.Position[12].Vel := 0;
   PRODUCT_TYPE[6].Motion.Gluing_Nozzle_Y.Position[12].Pos := 0.0;
   PRODUCT_TYPE[6].Motion.Gluing_Nozzle_Y.Position[12].Vel := 0;
   PRODUCT_TYPE[7].Motion.Gluing_Nozzle_Y.Position[12].Pos := 0.0;
   PRODUCT_TYPE[7].Motion.Gluing_Nozzle_Y.Position[12].Vel := 0;
   PRODUCT_TYPE[8].Motion.Gluing_Nozzle_Y.Position[12].Pos := 0.0;
   PRODUCT_TYPE[8].Motion.Gluing_Nozzle_Y.Position[12].Vel := 0;
   PRODUCT_TYPE[9].Motion.Gluing_Nozzle_Y.Position[12].Pos := 0.0;
   PRODUCT_TYPE[9].Motion.Gluing_Nozzle_Y.Position[12].Vel := 0;
   PRODUCT_TYPE[10].Motion.Gluing_Nozzle_Y.Position[12].Pos := 0.0;
   PRODUCT_TYPE[10].Motion.Gluing_Nozzle_Y.Position[12].Vel := 0;
   PRODUCT_TYPE[1].Motion.Gluing_Nozzle_Y.Position[13].Pos := 0.0;
   PRODUCT_TYPE[1].Motion.Gluing_Nozzle_Y.Position[13].Vel := 0;
   PRODUCT_TYPE[2].Motion.Gluing_Nozzle_Y.Position[13].Pos := 0.0;
   PRODUCT_TYPE[2].Motion.Gluing_Nozzle_Y.Position[13].Vel := 0;
   PRODUCT_TYPE[3].Motion.Gluing_Nozzle_Y.Position[13].Pos := 0.0;
   PRODUCT_TYPE[3].Motion.Gluing_Nozzle_Y.Position[13].Vel := 0;
   PRODUCT_TYPE[4].Motion.Gluing_Nozzle_Y.Position[13].Pos := 0.0;
   PRODUCT_TYPE[4].Motion.Gluing_Nozzle_Y.Position[13].Vel := 0;
   PRODUCT_TYPE[5].Motion.Gluing_Nozzle_Y.Position[13].Pos := 0.0;
   PRODUCT_TYPE[5].Motion.Gluing_Nozzle_Y.Position[13].Vel := 0;
   PRODUCT_TYPE[6].Motion.Gluing_Nozzle_Y.Position[13].Pos := 0.0;
   PRODUCT_TYPE[6].Motion.Gluing_Nozzle_Y.Position[13].Vel := 0;
   PRODUCT_TYPE[7].Motion.Gluing_Nozzle_Y.Position[13].Pos := 0.0;
   PRODUCT_TYPE[7].Motion.Gluing_Nozzle_Y.Position[13].Vel := 0;
   PRODUCT_TYPE[8].Motion.Gluing_Nozzle_Y.Position[13].Pos := 0.0;
   PRODUCT_TYPE[8].Motion.Gluing_Nozzle_Y.Position[13].Vel := 0;
   PRODUCT_TYPE[9].Motion.Gluing_Nozzle_Y.Position[13].Pos := 0.0;
   PRODUCT_TYPE[9].Motion.Gluing_Nozzle_Y.Position[13].Vel := 0;
   PRODUCT_TYPE[10].Motion.Gluing_Nozzle_Y.Position[13].Pos := 0.0;
   PRODUCT_TYPE[10].Motion.Gluing_Nozzle_Y.Position[13].Vel := 0;
   PRODUCT_TYPE[1].Motion.Gluing_Nozzle_Y.Position[14].Pos := 0.0;
   PRODUCT_TYPE[1].Motion.Gluing_Nozzle_Y.Position[14].Vel := 0;
   PRODUCT_TYPE[2].Motion.Gluing_Nozzle_Y.Position[14].Pos := 0.0;
   PRODUCT_TYPE[2].Motion.Gluing_Nozzle_Y.Position[14].Vel := 0;
   PRODUCT_TYPE[3].Motion.Gluing_Nozzle_Y.Position[14].Pos := 0.0;
   PRODUCT_TYPE[3].Motion.Gluing_Nozzle_Y.Position[14].Vel := 0;
   PRODUCT_TYPE[4].Motion.Gluing_Nozzle_Y.Position[14].Pos := 0.0;
   PRODUCT_TYPE[4].Motion.Gluing_Nozzle_Y.Position[14].Vel := 0;
   PRODUCT_TYPE[5].Motion.Gluing_Nozzle_Y.Position[14].Pos := 0.0;
   PRODUCT_TYPE[5].Motion.Gluing_Nozzle_Y.Position[14].Vel := 0;
   PRODUCT_TYPE[6].Motion.Gluing_Nozzle_Y.Position[14].Pos := 0.0;
   PRODUCT_TYPE[6].Motion.Gluing_Nozzle_Y.Position[14].Vel := 0;
   PRODUCT_TYPE[7].Motion.Gluing_Nozzle_Y.Position[14].Pos := 0.0;
   PRODUCT_TYPE[7].Motion.Gluing_Nozzle_Y.Position[14].Vel := 0;
   PRODUCT_TYPE[8].Motion.Gluing_Nozzle_Y.Position[14].Pos := 0.0;
   PRODUCT_TYPE[8].Motion.Gluing_Nozzle_Y.Position[14].Vel := 0;
   PRODUCT_TYPE[9].Motion.Gluing_Nozzle_Y.Position[14].Pos := 0.0;
   PRODUCT_TYPE[9].Motion.Gluing_Nozzle_Y.Position[14].Vel := 0;
   PRODUCT_TYPE[10].Motion.Gluing_Nozzle_Y.Position[14].Pos := 0.0;
   PRODUCT_TYPE[10].Motion.Gluing_Nozzle_Y.Position[14].Vel := 0;
   PRODUCT_TYPE[1].Motion.Gluing_Nozzle_Y.Position[15].Pos := 0.0;
   PRODUCT_TYPE[1].Motion.Gluing_Nozzle_Y.Position[15].Vel := 0;
   PRODUCT_TYPE[2].Motion.Gluing_Nozzle_Y.Position[15].Pos := 0.0;
   PRODUCT_TYPE[2].Motion.Gluing_Nozzle_Y.Position[15].Vel := 0;
   PRODUCT_TYPE[3].Motion.Gluing_Nozzle_Y.Position[15].Pos := 0.0;
   PRODUCT_TYPE[3].Motion.Gluing_Nozzle_Y.Position[15].Vel := 0;
   PRODUCT_TYPE[4].Motion.Gluing_Nozzle_Y.Position[15].Pos := 0.0;
   PRODUCT_TYPE[4].Motion.Gluing_Nozzle_Y.Position[15].Vel := 0;
   PRODUCT_TYPE[5].Motion.Gluing_Nozzle_Y.Position[15].Pos := 0.0;
   PRODUCT_TYPE[5].Motion.Gluing_Nozzle_Y.Position[15].Vel := 0;
   PRODUCT_TYPE[6].Motion.Gluing_Nozzle_Y.Position[15].Pos := 0.0;
   PRODUCT_TYPE[6].Motion.Gluing_Nozzle_Y.Position[15].Vel := 0;
   PRODUCT_TYPE[7].Motion.Gluing_Nozzle_Y.Position[15].Pos := 0.0;
   PRODUCT_TYPE[7].Motion.Gluing_Nozzle_Y.Position[15].Vel := 0;
   PRODUCT_TYPE[8].Motion.Gluing_Nozzle_Y.Position[15].Pos := 0.0;
   PRODUCT_TYPE[8].Motion.Gluing_Nozzle_Y.Position[15].Vel := 0;
   PRODUCT_TYPE[9].Motion.Gluing_Nozzle_Y.Position[15].Pos := 0.0;
   PRODUCT_TYPE[9].Motion.Gluing_Nozzle_Y.Position[15].Vel := 0;
   PRODUCT_TYPE[10].Motion.Gluing_Nozzle_Y.Position[15].Pos := 0.0;
   PRODUCT_TYPE[10].Motion.Gluing_Nozzle_Y.Position[15].Vel := 0;
   PRODUCT_TYPE[1].Motion.Gluing_Nozzle_Y.Position[16].Pos := 0.0;
   PRODUCT_TYPE[1].Motion.Gluing_Nozzle_Y.Position[16].Vel := 0;
   PRODUCT_TYPE[2].Motion.Gluing_Nozzle_Y.Position[16].Pos := 0.0;
   PRODUCT_TYPE[2].Motion.Gluing_Nozzle_Y.Position[16].Vel := 0;
   PRODUCT_TYPE[3].Motion.Gluing_Nozzle_Y.Position[16].Pos := 0.0;
   PRODUCT_TYPE[3].Motion.Gluing_Nozzle_Y.Position[16].Vel := 0;
   PRODUCT_TYPE[4].Motion.Gluing_Nozzle_Y.Position[16].Pos := 0.0;
   PRODUCT_TYPE[4].Motion.Gluing_Nozzle_Y.Position[16].Vel := 0;
   PRODUCT_TYPE[5].Motion.Gluing_Nozzle_Y.Position[16].Pos := 0.0;
   PRODUCT_TYPE[5].Motion.Gluing_Nozzle_Y.Position[16].Vel := 0;
   PRODUCT_TYPE[6].Motion.Gluing_Nozzle_Y.Position[16].Pos := 0.0;
   PRODUCT_TYPE[6].Motion.Gluing_Nozzle_Y.Position[16].Vel := 0;
   PRODUCT_TYPE[7].Motion.Gluing_Nozzle_Y.Position[16].Pos := 0.0;
   PRODUCT_TYPE[7].Motion.Gluing_Nozzle_Y.Position[16].Vel := 0;
   PRODUCT_TYPE[8].Motion.Gluing_Nozzle_Y.Position[16].Pos := 0.0;
   PRODUCT_TYPE[8].Motion.Gluing_Nozzle_Y.Position[16].Vel := 0;
   PRODUCT_TYPE[9].Motion.Gluing_Nozzle_Y.Position[16].Pos := 0.0;
   PRODUCT_TYPE[9].Motion.Gluing_Nozzle_Y.Position[16].Vel := 0;
   PRODUCT_TYPE[10].Motion.Gluing_Nozzle_Y.Position[16].Pos := 0.0;
   PRODUCT_TYPE[10].Motion.Gluing_Nozzle_Y.Position[16].Vel := 0;
   PRODUCT_TYPE[1].Motion.Gluing_Nozzle_Y.Position[17].Pos := 0.0;
   PRODUCT_TYPE[1].Motion.Gluing_Nozzle_Y.Position[17].Vel := 0;
   PRODUCT_TYPE[2].Motion.Gluing_Nozzle_Y.Position[17].Pos := 0.0;
   PRODUCT_TYPE[2].Motion.Gluing_Nozzle_Y.Position[17].Vel := 0;
   PRODUCT_TYPE[3].Motion.Gluing_Nozzle_Y.Position[17].Pos := 0.0;
   PRODUCT_TYPE[3].Motion.Gluing_Nozzle_Y.Position[17].Vel := 0;
   PRODUCT_TYPE[4].Motion.Gluing_Nozzle_Y.Position[17].Pos := 0.0;
   PRODUCT_TYPE[4].Motion.Gluing_Nozzle_Y.Position[17].Vel := 0;
   PRODUCT_TYPE[5].Motion.Gluing_Nozzle_Y.Position[17].Pos := 0.0;
   PRODUCT_TYPE[5].Motion.Gluing_Nozzle_Y.Position[17].Vel := 0;
   PRODUCT_TYPE[6].Motion.Gluing_Nozzle_Y.Position[17].Pos := 0.0;
   PRODUCT_TYPE[6].Motion.Gluing_Nozzle_Y.Position[17].Vel := 0;
   PRODUCT_TYPE[7].Motion.Gluing_Nozzle_Y.Position[17].Pos := 0.0;
   PRODUCT_TYPE[7].Motion.Gluing_Nozzle_Y.Position[17].Vel := 0;
   PRODUCT_TYPE[8].Motion.Gluing_Nozzle_Y.Position[17].Pos := 0.0;
   PRODUCT_TYPE[8].Motion.Gluing_Nozzle_Y.Position[17].Vel := 0;
   PRODUCT_TYPE[9].Motion.Gluing_Nozzle_Y.Position[17].Pos := 0.0;
   PRODUCT_TYPE[9].Motion.Gluing_Nozzle_Y.Position[17].Vel := 0;
   PRODUCT_TYPE[10].Motion.Gluing_Nozzle_Y.Position[17].Pos := 0.0;
   PRODUCT_TYPE[10].Motion.Gluing_Nozzle_Y.Position[17].Vel := 0;
   PRODUCT_TYPE[1].Motion.Gluing_Nozzle_Y.Position[18].Pos := 0.0;
   PRODUCT_TYPE[1].Motion.Gluing_Nozzle_Y.Position[18].Vel := 0;
   PRODUCT_TYPE[2].Motion.Gluing_Nozzle_Y.Position[18].Pos := 0.0;
   PRODUCT_TYPE[2].Motion.Gluing_Nozzle_Y.Position[18].Vel := 0;
   PRODUCT_TYPE[3].Motion.Gluing_Nozzle_Y.Position[18].Pos := 0.0;
   PRODUCT_TYPE[3].Motion.Gluing_Nozzle_Y.Position[18].Vel := 0;
   PRODUCT_TYPE[4].Motion.Gluing_Nozzle_Y.Position[18].Pos := 0.0;
   PRODUCT_TYPE[4].Motion.Gluing_Nozzle_Y.Position[18].Vel := 0;
   PRODUCT_TYPE[5].Motion.Gluing_Nozzle_Y.Position[18].Pos := 0.0;
   PRODUCT_TYPE[5].Motion.Gluing_Nozzle_Y.Position[18].Vel := 0;
   PRODUCT_TYPE[6].Motion.Gluing_Nozzle_Y.Position[18].Pos := 0.0;
   PRODUCT_TYPE[6].Motion.Gluing_Nozzle_Y.Position[18].Vel := 0;
   PRODUCT_TYPE[7].Motion.Gluing_Nozzle_Y.Position[18].Pos := 0.0;
   PRODUCT_TYPE[7].Motion.Gluing_Nozzle_Y.Position[18].Vel := 0;
   PRODUCT_TYPE[8].Motion.Gluing_Nozzle_Y.Position[18].Pos := 0.0;
   PRODUCT_TYPE[8].Motion.Gluing_Nozzle_Y.Position[18].Vel := 0;
   PRODUCT_TYPE[9].Motion.Gluing_Nozzle_Y.Position[18].Pos := 0.0;
   PRODUCT_TYPE[9].Motion.Gluing_Nozzle_Y.Position[18].Vel := 0;
   PRODUCT_TYPE[10].Motion.Gluing_Nozzle_Y.Position[18].Pos := 0.0;
   PRODUCT_TYPE[10].Motion.Gluing_Nozzle_Y.Position[18].Vel := 0;
   PRODUCT_TYPE[1].Motion.Gluing_Nozzle_Y.Position[19].Pos := 0.0;
   PRODUCT_TYPE[1].Motion.Gluing_Nozzle_Y.Position[19].Vel := 0;
   PRODUCT_TYPE[2].Motion.Gluing_Nozzle_Y.Position[19].Pos := 0.0;
   PRODUCT_TYPE[2].Motion.Gluing_Nozzle_Y.Position[19].Vel := 0;
   PRODUCT_TYPE[3].Motion.Gluing_Nozzle_Y.Position[19].Pos := 0.0;
   PRODUCT_TYPE[3].Motion.Gluing_Nozzle_Y.Position[19].Vel := 0;
   PRODUCT_TYPE[4].Motion.Gluing_Nozzle_Y.Position[19].Pos := 0.0;
   PRODUCT_TYPE[4].Motion.Gluing_Nozzle_Y.Position[19].Vel := 0;
   PRODUCT_TYPE[5].Motion.Gluing_Nozzle_Y.Position[19].Pos := 0.0;
   PRODUCT_TYPE[5].Motion.Gluing_Nozzle_Y.Position[19].Vel := 0;
   PRODUCT_TYPE[6].Motion.Gluing_Nozzle_Y.Position[19].Pos := 0.0;
   PRODUCT_TYPE[6].Motion.Gluing_Nozzle_Y.Position[19].Vel := 0;
   PRODUCT_TYPE[7].Motion.Gluing_Nozzle_Y.Position[19].Pos := 0.0;
   PRODUCT_TYPE[7].Motion.Gluing_Nozzle_Y.Position[19].Vel := 0;
   PRODUCT_TYPE[8].Motion.Gluing_Nozzle_Y.Position[19].Pos := 0.0;
   PRODUCT_TYPE[8].Motion.Gluing_Nozzle_Y.Position[19].Vel := 0;
   PRODUCT_TYPE[9].Motion.Gluing_Nozzle_Y.Position[19].Pos := 0.0;
   PRODUCT_TYPE[9].Motion.Gluing_Nozzle_Y.Position[19].Vel := 0;
   PRODUCT_TYPE[10].Motion.Gluing_Nozzle_Y.Position[19].Pos := 0.0;
   PRODUCT_TYPE[10].Motion.Gluing_Nozzle_Y.Position[19].Vel := 0;
   PRODUCT_TYPE[1].Motion.Gluing_Nozzle_Y.Position[20].Pos := 0.0;
   PRODUCT_TYPE[1].Motion.Gluing_Nozzle_Y.Position[20].Vel := 0;
   PRODUCT_TYPE[2].Motion.Gluing_Nozzle_Y.Position[20].Pos := 0.0;
   PRODUCT_TYPE[2].Motion.Gluing_Nozzle_Y.Position[20].Vel := 0;
   PRODUCT_TYPE[3].Motion.Gluing_Nozzle_Y.Position[20].Pos := 0.0;
   PRODUCT_TYPE[3].Motion.Gluing_Nozzle_Y.Position[20].Vel := 0;
   PRODUCT_TYPE[4].Motion.Gluing_Nozzle_Y.Position[20].Pos := 0.0;
   PRODUCT_TYPE[4].Motion.Gluing_Nozzle_Y.Position[20].Vel := 0;
   PRODUCT_TYPE[5].Motion.Gluing_Nozzle_Y.Position[20].Pos := 0.0;
